   S704_WELD_BUFF_DATA31.RBT2_BT_CODE_NO := W#16#0;
   S704_WELD_BUFF_DATA31.RBT2_WELD_COUNT := W#16#0;
   S704_WELD_BUFF_DATA31.RBT3_BT_CODE_NO := W#16#0;
   S704_WELD_BUFF_DATA31.RBT3_WELD_COUNT := W#16#0;
   S704_WELD_BUFF_DATA31.RBT4_BT_CODE_NO := W#16#0;
   S704_WELD_BUFF_DATA31.RBT4_WELD_COUNT := W#16#0;
   S704_WELD_BUFF_DATA31.RBT5_BT_CODE_NO := W#16#0;
   S704_WELD_BUFF_DATA31.RBT5_WELD_COUNT := W#16#0;
   S704_WELD_BUFF_DATA31.RBT6_BT_CODE_NO := W#16#0;
   S704_WELD_BUFF_DATA31.RBT6_WELD_COUNT := W#16#0;
   S704_WELD_BUFF_DATA31.RBT7_BT_CODE_NO := W#16#0;
   S704_WELD_BUFF_DATA31.RBT7_WELD_COUNT := W#16#0;
   S704_WELD_BUFF_DATA31.RBT8_BT_CODE_NO := W#16#0;
   S704_WELD_BUFF_DATA31.RBT8_WELD_COUNT := W#16#0;
   S704_WELD_BUFF_DATA31.RBT9_BT_CODE_NO := W#16#0;
   S704_WELD_BUFF_DATA31.RBT9_WELD_COUNT := W#16#0;
   S704_WELD_BUFF_DATA31.RBT10_BT_CODE_NO := W#16#0;
   S704_WELD_BUFF_DATA31.RBT10_WELD_COUNT := W#16#0;
   S704_WELD_BUFF_DATA31.RBT11_BT_CODE_NO := W#16#0;
   S704_WELD_BUFF_DATA31.RBT11_WELD_COUNT := W#16#0;
   S704_WELD_BUFF_DATA31.RBT12_BT_CODE_NO := W#16#0;
   S704_WELD_BUFF_DATA31.RBT12_WELD_COUNT := W#16#0;
   S704_WELD_BUFF_DATA31.RBT13_BT_CODE_NO := W#16#0;
   S704_WELD_BUFF_DATA31.RBT13_WELD_COUNT := W#16#0;
   S704_WELD_BUFF_DATA31.RBT14_BT_CODE_NO := W#16#0;
   S704_WELD_BUFF_DATA31.RBT14_WELD_COUNT := W#16#0;
   S704_WELD_BUFF_DATA31.RBT15_BT_CODE_NO := W#16#0;
   S704_WELD_BUFF_DATA31.RBT15_WELD_COUNT := W#16#0;
   S704_WELD_BUFF_DATA31.RBT16_BT_CODE_NO := W#16#0;
   S704_WELD_BUFF_DATA31.RBT16_WELD_COUNT := W#16#0;
   S704_WELD_BUFF_DATA31.RBT17_BT_CODE_NO := W#16#0;
   S704_WELD_BUFF_DATA31.RBT17_WELD_COUNT := W#16#0;
   S704_WELD_BUFF_DATA31.RBT18_BT_CODE_NO := W#16#0;
   S704_WELD_BUFF_DATA31.RBT18_WELD_COUNT := W#16#0;
   S704_WELD_BUFF_DATA31.RBT19_BT_CODE_NO := W#16#0;
   S704_WELD_BUFF_DATA31.RBT19_WELD_COUNT := W#16#0;
   S704_WELD_BUFF_DATA31.RBT20_BT_CODE_NO := W#16#0;
   S704_WELD_BUFF_DATA31.RBT20_WELD_COUNT := W#16#0;
   S704_WELD_BUFF_DATA31.RBT21_BT_CODE_NO := W#16#0;
   S704_WELD_BUFF_DATA31.RBT21_WELD_COUNT := W#16#0;
   S704_WELD_BUFF_DATA31.RBT22_BT_CODE_NO := W#16#0;
   S704_WELD_BUFF_DATA31.RBT22_WELD_COUNT := W#16#0;
   S704_WELD_BUFF_DATA31.RBT23_BT_CODE_NO := W#16#0;
   S704_WELD_BUFF_DATA31.RBT23_WELD_COUNT := W#16#0;
   S704_WELD_BUFF_DATA31.RBT24_BT_CODE_NO := W#16#0;
   S704_WELD_BUFF_DATA31.RBT24_WELD_COUNT := W#16#0;
   S704_WELD_BUFF_DATA31.WELD_DETERMINES_RESULT := W#16#0;
   S704_WELD_BUFF_DATA31.WELD_CHECK_SUM := W#16#0;
   S704_WELD_BUFF_DATA31.SPARE1 := W#16#0;
   S704_WELD_BUFF_DATA41.STATION_MAIN := W#16#0;
   S704_WELD_BUFF_DATA41.DISTINCTION_LH_RH := W#16#0;
   S704_WELD_BUFF_DATA41.STAION_NUMBER := W#16#0;
   S704_WELD_BUFF_DATA41.VIN_NUMBER1 := W#16#0;
   S704_WELD_BUFF_DATA41.VIN_NUMBER2 := W#16#0;
   S704_WELD_BUFF_DATA41.VIN_NUMBER3 := W#16#0;
   S704_WELD_BUFF_DATA41.VIN_NUMBER4 := W#16#0;
   S704_WELD_BUFF_DATA41.SEQ_NUMBER1 := W#16#0;
   S704_WELD_BUFF_DATA41.SEQ_NUMBER2 := W#16#0;
   S704_WELD_BUFF_DATA41.RBT1_BT_CODE_NO := W#16#0;
   S704_WELD_BUFF_DATA41.RBT1_WELD_COUNT := W#16#0;
   S704_WELD_BUFF_DATA41.RBT2_BT_CODE_NO := W#16#0;
   S704_WELD_BUFF_DATA41.RBT2_WELD_COUNT := W#16#0;
   S704_WELD_BUFF_DATA41.RBT3_BT_CODE_NO := W#16#0;
   S704_WELD_BUFF_DATA41.RBT3_WELD_COUNT := W#16#0;
   S704_WELD_BUFF_DATA41.RBT4_BT_CODE_NO := W#16#0;
   S704_WELD_BUFF_DATA41.RBT4_WELD_COUNT := W#16#0;
   S704_WELD_BUFF_DATA41.RBT5_BT_CODE_NO := W#16#0;
   S704_WELD_BUFF_DATA41.RBT5_WELD_COUNT := W#16#0;
   S704_WELD_BUFF_DATA41.RBT6_BT_CODE_NO := W#16#0;
   S704_WELD_BUFF_DATA41.RBT6_WELD_COUNT := W#16#0;
   S704_WELD_BUFF_DATA41.RBT7_BT_CODE_NO := W#16#0;
   S704_WELD_BUFF_DATA41.RBT7_WELD_COUNT := W#16#0;
   S704_WELD_BUFF_DATA41.RBT8_BT_CODE_NO := W#16#0;
   S704_WELD_BUFF_DATA41.RBT8_WELD_COUNT := W#16#0;
   S704_WELD_BUFF_DATA41.RBT9_BT_CODE_NO := W#16#0;
   S704_WELD_BUFF_DATA41.RBT9_WELD_COUNT := W#16#0;
   S704_WELD_BUFF_DATA41.RBT10_BT_CODE_NO := W#16#0;
   S704_WELD_BUFF_DATA41.RBT10_WELD_COUNT := W#16#0;
   S704_WELD_BUFF_DATA41.RBT11_BT_CODE_NO := W#16#0;
   S704_WELD_BUFF_DATA41.RBT11_WELD_COUNT := W#16#0;
   S704_WELD_BUFF_DATA41.RBT12_BT_CODE_NO := W#16#0;
   S704_WELD_BUFF_DATA41.RBT12_WELD_COUNT := W#16#0;
   S704_WELD_BUFF_DATA41.RBT13_BT_CODE_NO := W#16#0;
   S704_WELD_BUFF_DATA41.RBT13_WELD_COUNT := W#16#0;
   S704_WELD_BUFF_DATA41.RBT14_BT_CODE_NO := W#16#0;
   S704_WELD_BUFF_DATA41.RBT14_WELD_COUNT := W#16#0;
   S704_WELD_BUFF_DATA41.RBT15_BT_CODE_NO := W#16#0;
   S704_WELD_BUFF_DATA41.RBT15_WELD_COUNT := W#16#0;
   S704_WELD_BUFF_DATA41.RBT16_BT_CODE_NO := W#16#0;
   S704_WELD_BUFF_DATA41.RBT16_WELD_COUNT := W#16#0;
   S704_WELD_BUFF_DATA41.RBT17_BT_CODE_NO := W#16#0;
   S704_WELD_BUFF_DATA41.RBT17_WELD_COUNT := W#16#0;
   S704_WELD_BUFF_DATA41.RBT18_BT_CODE_NO := W#16#0;
   S704_WELD_BUFF_DATA41.RBT18_WELD_COUNT := W#16#0;
   S704_WELD_BUFF_DATA41.RBT19_BT_CODE_NO := W#16#0;
   S704_WELD_BUFF_DATA41.RBT19_WELD_COUNT := W#16#0;
   S704_WELD_BUFF_DATA41.RBT20_BT_CODE_NO := W#16#0;
   S704_WELD_BUFF_DATA41.RBT20_WELD_COUNT := W#16#0;
   S704_WELD_BUFF_DATA41.RBT21_BT_CODE_NO := W#16#0;
   S704_WELD_BUFF_DATA41.RBT21_WELD_COUNT := W#16#0;
   S704_WELD_BUFF_DATA41.RBT22_BT_CODE_NO := W#16#0;
   S704_WELD_BUFF_DATA41.RBT22_WELD_COUNT := W#16#0;
   S704_WELD_BUFF_DATA41.RBT23_BT_CODE_NO := W#16#0;
   S704_WELD_BUFF_DATA41.RBT23_WELD_COUNT := W#16#0;
   S704_WELD_BUFF_DATA41.RBT24_BT_CODE_NO := W#16#0;
   S704_WELD_BUFF_DATA41.RBT24_WELD_COUNT := W#16#0;
   S704_WELD_BUFF_DATA41.WELD_DETERMINES_RESULT := W#16#0;
   S704_WELD_BUFF_DATA41.WELD_CHECK_SUM := W#16#0;
   S704_WELD_BUFF_DATA41.SPARE1 := W#16#0;
   S704_WELD_BUFF_DATA51.STATION_MAIN := W#16#0;
   S704_WELD_BUFF_DATA51.DISTINCTION_LH_RH := W#16#0;
   S704_WELD_BUFF_DATA51.STAION_NUMBER := W#16#0;
   S704_WELD_BUFF_DATA51.VIN_NUMBER1 := W#16#0;
   S704_WELD_BUFF_DATA51.VIN_NUMBER2 := W#16#0;
   S704_WELD_BUFF_DATA51.VIN_NUMBER3 := W#16#0;
   S704_WELD_BUFF_DATA51.VIN_NUMBER4 := W#16#0;
   S704_WELD_BUFF_DATA51.SEQ_NUMBER1 := W#16#0;
   S704_WELD_BUFF_DATA51.SEQ_NUMBER2 := W#16#0;
   S704_WELD_BUFF_DATA51.RBT1_BT_CODE_NO := W#16#0;
   S704_WELD_BUFF_DATA51.RBT1_WELD_COUNT := W#16#0;
   S704_WELD_BUFF_DATA51.RBT2_BT_CODE_NO := W#16#0;
   S704_WELD_BUFF_DATA51.RBT2_WELD_COUNT := W#16#0;
   S704_WELD_BUFF_DATA51.RBT3_BT_CODE_NO := W#16#0;
   S704_WELD_BUFF_DATA51.RBT3_WELD_COUNT := W#16#0;
   S704_WELD_BUFF_DATA51.RBT4_BT_CODE_NO := W#16#0;
   S704_WELD_BUFF_DATA51.RBT4_WELD_COUNT := W#16#0;
   S704_WELD_BUFF_DATA51.RBT5_BT_CODE_NO := W#16#0;
   S704_WELD_BUFF_DATA51.RBT5_WELD_COUNT := W#16#0;
   S704_WELD_BUFF_DATA51.RBT6_BT_CODE_NO := W#16#0;
   S704_WELD_BUFF_DATA51.RBT6_WELD_COUNT := W#16#0;
   S704_WELD_BUFF_DATA51.RBT7_BT_CODE_NO := W#16#0;
   S704_WELD_BUFF_DATA51.RBT7_WELD_COUNT := W#16#0;
   S704_WELD_BUFF_DATA51.RBT8_BT_CODE_NO := W#16#0;
   S704_WELD_BUFF_DATA51.RBT8_WELD_COUNT := W#16#0;
   S704_WELD_BUFF_DATA51.RBT9_BT_CODE_NO := W#16#0;
   S704_WELD_BUFF_DATA51.RBT9_WELD_COUNT := W#16#0;
   S704_WELD_BUFF_DATA51.RBT10_BT_CODE_NO := W#16#0;
   S704_WELD_BUFF_DATA51.RBT10_WELD_COUNT := W#16#0;
   S704_WELD_BUFF_DATA51.RBT11_BT_CODE_NO := W#16#0;
   S704_WELD_BUFF_DATA51.RBT11_WELD_COUNT := W#16#0;
   S704_WELD_BUFF_DATA51.RBT12_BT_CODE_NO := W#16#0;
   S704_WELD_BUFF_DATA51.RBT12_WELD_COUNT := W#16#0;
   S704_WELD_BUFF_DATA51.RBT13_BT_CODE_NO := W#16#0;
   S704_WELD_BUFF_DATA51.RBT13_WELD_COUNT := W#16#0;
   S704_WELD_BUFF_DATA51.RBT14_BT_CODE_NO := W#16#0;
   S704_WELD_BUFF_DATA51.RBT14_WELD_COUNT := W#16#0;
   S704_WELD_BUFF_DATA51.RBT15_BT_CODE_NO := W#16#0;
   S704_WELD_BUFF_DATA51.RBT15_WELD_COUNT := W#16#0;
   S704_WELD_BUFF_DATA51.RBT16_BT_CODE_NO := W#16#0;
   S704_WELD_BUFF_DATA51.RBT16_WELD_COUNT := W#16#0;
   S704_WELD_BUFF_DATA51.RBT17_BT_CODE_NO := W#16#0;
   S704_WELD_BUFF_DATA51.RBT17_WELD_COUNT := W#16#0;
   S704_WELD_BUFF_DATA51.RBT18_BT_CODE_NO := W#16#0;
   S704_WELD_BUFF_DATA51.RBT18_WELD_COUNT := W#16#0;
   S704_WELD_BUFF_DATA51.RBT19_BT_CODE_NO := W#16#0;
   S704_WELD_BUFF_DATA51.RBT19_WELD_COUNT := W#16#0;
   S704_WELD_BUFF_DATA51.RBT20_BT_CODE_NO := W#16#0;
   S704_WELD_BUFF_DATA51.RBT20_WELD_COUNT := W#16#0;
   S704_WELD_BUFF_DATA51.RBT21_BT_CODE_NO := W#16#0;
   S704_WELD_BUFF_DATA51.RBT21_WELD_COUNT := W#16#0;
   S704_WELD_BUFF_DATA51.RBT22_BT_CODE_NO := W#16#0;
   S704_WELD_BUFF_DATA51.RBT22_WELD_COUNT := W#16#0;
   S704_WELD_BUFF_DATA51.RBT23_BT_CODE_NO := W#16#0;
   S704_WELD_BUFF_DATA51.RBT23_WELD_COUNT := W#16#0;
   S704_WELD_BUFF_DATA51.RBT24_BT_CODE_NO := W#16#0;
   S704_WELD_BUFF_DATA51.RBT24_WELD_COUNT := W#16#0;
   S704_WELD_BUFF_DATA51.WELD_DETERMINES_RESULT := W#16#0;
   S704_WELD_BUFF_DATA51.WELD_CHECK_SUM := W#16#0;
   S704_WELD_BUFF_DATA51.SPARE1 := W#16#0;
   S704_WELD_BUFF_DATA61.STATION_MAIN := W#16#0;
   S704_WELD_BUFF_DATA61.DISTINCTION_LH_RH := W#16#0;
   S704_WELD_BUFF_DATA61.STAION_NUMBER := W#16#0;
   S704_WELD_BUFF_DATA61.VIN_NUMBER1 := W#16#0;
   S704_WELD_BUFF_DATA61.VIN_NUMBER2 := W#16#0;
   S704_WELD_BUFF_DATA61.VIN_NUMBER3 := W#16#0;
   S704_WELD_BUFF_DATA61.VIN_NUMBER4 := W#16#0;
   S704_WELD_BUFF_DATA61.SEQ_NUMBER1 := W#16#0;
   S704_WELD_BUFF_DATA61.SEQ_NUMBER2 := W#16#0;
   S704_WELD_BUFF_DATA61.RBT1_BT_CODE_NO := W#16#0;
   S704_WELD_BUFF_DATA61.RBT1_WELD_COUNT := W#16#0;
   S704_WELD_BUFF_DATA61.RBT2_BT_CODE_NO := W#16#0;
   S704_WELD_BUFF_DATA61.RBT2_WELD_COUNT := W#16#0;
   S704_WELD_BUFF_DATA61.RBT3_BT_CODE_NO := W#16#0;
   S704_WELD_BUFF_DATA61.RBT3_WELD_COUNT := W#16#0;
   S704_WELD_BUFF_DATA61.RBT4_BT_CODE_NO := W#16#0;
   S704_WELD_BUFF_DATA61.RBT4_WELD_COUNT := W#16#0;
   S704_WELD_BUFF_DATA61.RBT5_BT_CODE_NO := W#16#0;
   S704_WELD_BUFF_DATA61.RBT5_WELD_COUNT := W#16#0;
   S704_WELD_BUFF_DATA61.RBT6_BT_CODE_NO := W#16#0;
   S704_WELD_BUFF_DATA61.RBT6_WELD_COUNT := W#16#0;
   S704_WELD_BUFF_DATA61.RBT7_BT_CODE_NO := W#16#0;
   S704_WELD_BUFF_DATA61.RBT7_WELD_COUNT := W#16#0;
   S704_WELD_BUFF_DATA61.RBT8_BT_CODE_NO := W#16#0;
   S704_WELD_BUFF_DATA61.RBT8_WELD_COUNT := W#16#0;
   S704_WELD_BUFF_DATA61.RBT9_BT_CODE_NO := W#16#0;
   S704_WELD_BUFF_DATA61.RBT9_WELD_COUNT := W#16#0;
   S704_WELD_BUFF_DATA61.RBT10_BT_CODE_NO := W#16#0;
   S704_WELD_BUFF_DATA61.RBT10_WELD_COUNT := W#16#0;
   S704_WELD_BUFF_DATA61.RBT11_BT_CODE_NO := W#16#0;
   S704_WELD_BUFF_DATA61.RBT11_WELD_COUNT := W#16#0;
   S704_WELD_BUFF_DATA61.RBT12_BT_CODE_NO := W#16#0;
   S704_WELD_BUFF_DATA61.RBT12_WELD_COUNT := W#16#0;
   S704_WELD_BUFF_DATA61.RBT13_BT_CODE_NO := W#16#0;
   S704_WELD_BUFF_DATA61.RBT13_WELD_COUNT := W#16#0;
   S704_WELD_BUFF_DATA61.RBT14_BT_CODE_NO := W#16#0;
   S704_WELD_BUFF_DATA61.RBT14_WELD_COUNT := W#16#0;
   S704_WELD_BUFF_DATA61.RBT15_BT_CODE_NO := W#16#0;
   S704_WELD_BUFF_DATA61.RBT15_WELD_COUNT := W#16#0;
   S704_WELD_BUFF_DATA61.RBT16_BT_CODE_NO := W#16#0;
   S704_WELD_BUFF_DATA61.RBT16_WELD_COUNT := W#16#0;
   S704_WELD_BUFF_DATA61.RBT17_BT_CODE_NO := W#16#0;
   S704_WELD_BUFF_DATA61.RBT17_WELD_COUNT := W#16#0;
   S704_WELD_BUFF_DATA61.RBT18_BT_CODE_NO := W#16#0;
   S704_WELD_BUFF_DATA61.RBT18_WELD_COUNT := W#16#0;
   S704_WELD_BUFF_DATA61.RBT19_BT_CODE_NO := W#16#0;
   S704_WELD_BUFF_DATA61.RBT19_WELD_COUNT := W#16#0;
   S704_WELD_BUFF_DATA61.RBT20_BT_CODE_NO := W#16#0;
   S704_WELD_BUFF_DATA61.RBT20_WELD_COUNT := W#16#0;
   S704_WELD_BUFF_DATA61.RBT21_BT_CODE_NO := W#16#0;
   S704_WELD_BUFF_DATA61.RBT21_WELD_COUNT := W#16#0;
   S704_WELD_BUFF_DATA61.RBT22_BT_CODE_NO := W#16#0;
   S704_WELD_BUFF_DATA61.RBT22_WELD_COUNT := W#16#0;
   S704_WELD_BUFF_DATA61.RBT23_BT_CODE_NO := W#16#0;
   S704_WELD_BUFF_DATA61.RBT23_WELD_COUNT := W#16#0;
   S704_WELD_BUFF_DATA61.RBT24_BT_CODE_NO := W#16#0;
   S704_WELD_BUFF_DATA61.RBT24_WELD_COUNT := W#16#0;
   S704_WELD_BUFF_DATA61.WELD_DETERMINES_RESULT := W#16#0;
   S704_WELD_BUFF_DATA61.WELD_CHECK_SUM := W#16#0;
   S704_WELD_BUFF_DATA61.SPARE1 := W#16#0;
   S704_WELD_BUFF_DATA71.STATION_MAIN := W#16#0;
   S704_WELD_BUFF_DATA71.DISTINCTION_LH_RH := W#16#0;
   S704_WELD_BUFF_DATA71.STAION_NUMBER := W#16#0;
   S704_WELD_BUFF_DATA71.VIN_NUMBER1 := W#16#0;
   S704_WELD_BUFF_DATA71.VIN_NUMBER2 := W#16#0;
   S704_WELD_BUFF_DATA71.VIN_NUMBER3 := W#16#0;
   S704_WELD_BUFF_DATA71.VIN_NUMBER4 := W#16#0;
   S704_WELD_BUFF_DATA71.SEQ_NUMBER1 := W#16#0;
   S704_WELD_BUFF_DATA71.SEQ_NUMBER2 := W#16#0;
   S704_WELD_BUFF_DATA71.RBT1_BT_CODE_NO := W#16#0;
   S704_WELD_BUFF_DATA71.RBT1_WELD_COUNT := W#16#0;
   S704_WELD_BUFF_DATA71.RBT2_BT_CODE_NO := W#16#0;
   S704_WELD_BUFF_DATA71.RBT2_WELD_COUNT := W#16#0;
   S704_WELD_BUFF_DATA71.RBT3_BT_CODE_NO := W#16#0;
   S704_WELD_BUFF_DATA71.RBT3_WELD_COUNT := W#16#0;
   S704_WELD_BUFF_DATA71.RBT4_BT_CODE_NO := W#16#0;
   S704_WELD_BUFF_DATA71.RBT4_WELD_COUNT := W#16#0;
   S704_WELD_BUFF_DATA71.RBT5_BT_CODE_NO := W#16#0;
   S704_WELD_BUFF_DATA71.RBT5_WELD_COUNT := W#16#0;
   S704_WELD_BUFF_DATA71.RBT6_BT_CODE_NO := W#16#0;
   S704_WELD_BUFF_DATA71.RBT6_WELD_COUNT := W#16#0;
   S704_WELD_BUFF_DATA71.RBT7_BT_CODE_NO := W#16#0;
   S704_WELD_BUFF_DATA71.RBT7_WELD_COUNT := W#16#0;
   S704_WELD_BUFF_DATA71.RBT8_BT_CODE_NO := W#16#0;
   S704_WELD_BUFF_DATA71.RBT8_WELD_COUNT := W#16#0;
   S704_WELD_BUFF_DATA71.RBT9_BT_CODE_NO := W#16#0;
   S704_WELD_BUFF_DATA71.RBT9_WELD_COUNT := W#16#0;
   S704_WELD_BUFF_DATA71.RBT10_BT_CODE_NO := W#16#0;
   S704_WELD_BUFF_DATA71.RBT10_WELD_COUNT := W#16#0;
   S704_WELD_BUFF_DATA71.RBT11_BT_CODE_NO := W#16#0;
   S704_WELD_BUFF_DATA71.RBT11_WELD_COUNT := W#16#0;
   S704_WELD_BUFF_DATA71.RBT12_BT_CODE_NO := W#16#0;
   S704_WELD_BUFF_DATA71.RBT12_WELD_COUNT := W#16#0;
   S704_WELD_BUFF_DATA71.RBT13_BT_CODE_NO := W#16#0;
   S704_WELD_BUFF_DATA71.RBT13_WELD_COUNT := W#16#0;
   S704_WELD_BUFF_DATA71.RBT14_BT_CODE_NO := W#16#0;
   S704_WELD_BUFF_DATA71.RBT14_WELD_COUNT := W#16#0;
   S704_WELD_BUFF_DATA71.RBT15_BT_CODE_NO := W#16#0;
   S704_WELD_BUFF_DATA71.RBT15_WELD_COUNT := W#16#0;
   S704_WELD_BUFF_DATA71.RBT16_BT_CODE_NO := W#16#0;
   S704_WELD_BUFF_DATA71.RBT16_WELD_COUNT := W#16#0;
   S704_WELD_BUFF_DATA71.RBT17_BT_CODE_NO := W#16#0;
   S704_WELD_BUFF_DATA71.RBT17_WELD_COUNT := W#16#0;
   S704_WELD_BUFF_DATA71.RBT18_BT_CODE_NO := W#16#0;
   S704_WELD_BUFF_DATA71.RBT18_WELD_COUNT := W#16#0;
   S704_WELD_BUFF_DATA71.RBT19_BT_CODE_NO := W#16#0;
   S704_WELD_BUFF_DATA71.RBT19_WELD_COUNT := W#16#0;
   S704_WELD_BUFF_DATA71.RBT20_BT_CODE_NO := W#16#0;
   S704_WELD_BUFF_DATA71.RBT20_WELD_COUNT := W#16#0;
   S704_WELD_BUFF_DATA71.RBT21_BT_CODE_NO := W#16#0;
   S704_WELD_BUFF_DATA71.RBT21_WELD_COUNT := W#16#0;
   S704_WELD_BUFF_DATA71.RBT22_BT_CODE_NO := W#16#0;
   S704_WELD_BUFF_DATA71.RBT22_WELD_COUNT := W#16#0;
   S704_WELD_BUFF_DATA71.RBT23_BT_CODE_NO := W#16#0;
   S704_WELD_BUFF_DATA71.RBT23_WELD_COUNT := W#16#0;
   S704_WELD_BUFF_DATA71.RBT24_BT_CODE_NO := W#16#0;
   S704_WELD_BUFF_DATA71.RBT24_WELD_COUNT := W#16#0;
   S704_WELD_BUFF_DATA71.WELD_DETERMINES_RESULT := W#16#0;
   S704_WELD_BUFF_DATA71.WELD_CHECK_SUM := W#16#0;
   S704_WELD_BUFF_DATA71.SPARE1 := W#16#0;
   S704_WELD_BUFF_DATA81.STATION_MAIN := W#16#0;
   S704_WELD_BUFF_DATA81.DISTINCTION_LH_RH := W#16#0;
   S704_WELD_BUFF_DATA81.STAION_NUMBER := W#16#0;
   S704_WELD_BUFF_DATA81.VIN_NUMBER1 := W#16#0;
   S704_WELD_BUFF_DATA81.VIN_NUMBER2 := W#16#0;
   S704_WELD_BUFF_DATA81.VIN_NUMBER3 := W#16#0;
   S704_WELD_BUFF_DATA81.VIN_NUMBER4 := W#16#0;
   S704_WELD_BUFF_DATA81.SEQ_NUMBER1 := W#16#0;
   S704_WELD_BUFF_DATA81.SEQ_NUMBER2 := W#16#0;
   S704_WELD_BUFF_DATA81.RBT1_BT_CODE_NO := W#16#0;
   S704_WELD_BUFF_DATA81.RBT1_WELD_COUNT := W#16#0;
   S704_WELD_BUFF_DATA81.RBT2_BT_CODE_NO := W#16#0;
   S704_WELD_BUFF_DATA81.RBT2_WELD_COUNT := W#16#0;
   S704_WELD_BUFF_DATA81.RBT3_BT_CODE_NO := W#16#0;
   S704_WELD_BUFF_DATA81.RBT3_WELD_COUNT := W#16#0;
   S704_WELD_BUFF_DATA81.RBT4_BT_CODE_NO := W#16#0;
   S704_WELD_BUFF_DATA81.RBT4_WELD_COUNT := W#16#0;
   S704_WELD_BUFF_DATA81.RBT5_BT_CODE_NO := W#16#0;
   S704_WELD_BUFF_DATA81.RBT5_WELD_COUNT := W#16#0;
   S704_WELD_BUFF_DATA81.RBT6_BT_CODE_NO := W#16#0;
   S704_WELD_BUFF_DATA81.RBT6_WELD_COUNT := W#16#0;
   S704_WELD_BUFF_DATA81.RBT7_BT_CODE_NO := W#16#0;
   S704_WELD_BUFF_DATA81.RBT7_WELD_COUNT := W#16#0;
   S704_WELD_BUFF_DATA81.RBT8_BT_CODE_NO := W#16#0;
   S704_WELD_BUFF_DATA81.RBT8_WELD_COUNT := W#16#0;
   S704_WELD_BUFF_DATA81.RBT9_BT_CODE_NO := W#16#0;
   S704_WELD_BUFF_DATA81.RBT9_WELD_COUNT := W#16#0;
   S704_WELD_BUFF_DATA81.RBT10_BT_CODE_NO := W#16#0;
   S704_WELD_BUFF_DATA81.RBT10_WELD_COUNT := W#16#0;
   S704_WELD_BUFF_DATA81.RBT11_BT_CODE_NO := W#16#0;
   S704_WELD_BUFF_DATA81.RBT11_WELD_COUNT := W#16#0;
   S704_WELD_BUFF_DATA81.RBT12_BT_CODE_NO := W#16#0;
   S704_WELD_BUFF_DATA81.RBT12_WELD_COUNT := W#16#0;
   S704_WELD_BUFF_DATA81.RBT13_BT_CODE_NO := W#16#0;
   S704_WELD_BUFF_DATA81.RBT13_WELD_COUNT := W#16#0;
   S704_WELD_BUFF_DATA81.RBT14_BT_CODE_NO := W#16#0;
   S704_WELD_BUFF_DATA81.RBT14_WELD_COUNT := W#16#0;
   S704_WELD_BUFF_DATA81.RBT15_BT_CODE_NO := W#16#0;
   S704_WELD_BUFF_DATA81.RBT15_WELD_COUNT := W#16#0;
   S704_WELD_BUFF_DATA81.RBT16_BT_CODE_NO := W#16#0;
   S704_WELD_BUFF_DATA81.RBT16_WELD_COUNT := W#16#0;
   S704_WELD_BUFF_DATA81.RBT17_BT_CODE_NO := W#16#0;
   S704_WELD_BUFF_DATA81.RBT17_WELD_COUNT := W#16#0;
   S704_WELD_BUFF_DATA81.RBT18_BT_CODE_NO := W#16#0;
   S704_WELD_BUFF_DATA81.RBT18_WELD_COUNT := W#16#0;
   S704_WELD_BUFF_DATA81.RBT19_BT_CODE_NO := W#16#0;
   S704_WELD_BUFF_DATA81.RBT19_WELD_COUNT := W#16#0;
   S704_WELD_BUFF_DATA81.RBT20_BT_CODE_NO := W#16#0;
   S704_WELD_BUFF_DATA81.RBT20_WELD_COUNT := W#16#0;
   S704_WELD_BUFF_DATA81.RBT21_BT_CODE_NO := W#16#0;
   S704_WELD_BUFF_DATA81.RBT21_WELD_COUNT := W#16#0;
   S704_WELD_BUFF_DATA81.RBT22_BT_CODE_NO := W#16#0;
   S704_WELD_BUFF_DATA81.RBT22_WELD_COUNT := W#16#0;
   S704_WELD_BUFF_DATA81.RBT23_BT_CODE_NO := W#16#0;
   S704_WELD_BUFF_DATA81.RBT23_WELD_COUNT := W#16#0;
   S704_WELD_BUFF_DATA81.RBT24_BT_CODE_NO := W#16#0;
   S704_WELD_BUFF_DATA81.RBT24_WELD_COUNT := W#16#0;
   S704_WELD_BUFF_DATA81.WELD_DETERMINES_RESULT := W#16#0;
   S704_WELD_BUFF_DATA81.WELD_CHECK_SUM := W#16#0;
   S704_WELD_BUFF_DATA81.SPARE1 := W#16#0;
   S704_WELD_BUFF_DATA91.STATION_MAIN := W#16#0;
   S704_WELD_BUFF_DATA91.DISTINCTION_LH_RH := W#16#0;
   S704_WELD_BUFF_DATA91.STAION_NUMBER := W#16#0;
   S704_WELD_BUFF_DATA91.VIN_NUMBER1 := W#16#0;
   S704_WELD_BUFF_DATA91.VIN_NUMBER2 := W#16#0;
   S704_WELD_BUFF_DATA91.VIN_NUMBER3 := W#16#0;
   S704_WELD_BUFF_DATA91.VIN_NUMBER4 := W#16#0;
   S704_WELD_BUFF_DATA91.SEQ_NUMBER1 := W#16#0;
   S704_WELD_BUFF_DATA91.SEQ_NUMBER2 := W#16#0;
   S704_WELD_BUFF_DATA91.RBT1_BT_CODE_NO := W#16#0;
   S704_WELD_BUFF_DATA91.RBT1_WELD_COUNT := W#16#0;
   S704_WELD_BUFF_DATA91.RBT2_BT_CODE_NO := W#16#0;
   S704_WELD_BUFF_DATA91.RBT2_WELD_COUNT := W#16#0;
   S704_WELD_BUFF_DATA91.RBT3_BT_CODE_NO := W#16#0;
   S704_WELD_BUFF_DATA91.RBT3_WELD_COUNT := W#16#0;
   S704_WELD_BUFF_DATA91.RBT4_BT_CODE_NO := W#16#0;
   S704_WELD_BUFF_DATA91.RBT4_WELD_COUNT := W#16#0;
   S704_WELD_BUFF_DATA91.RBT5_BT_CODE_NO := W#16#0;
   S704_WELD_BUFF_DATA91.RBT5_WELD_COUNT := W#16#0;
   S704_WELD_BUFF_DATA91.RBT6_BT_CODE_NO := W#16#0;
   S704_WELD_BUFF_DATA91.RBT6_WELD_COUNT := W#16#0;
   S704_WELD_BUFF_DATA91.RBT7_BT_CODE_NO := W#16#0;
   S704_WELD_BUFF_DATA91.RBT7_WELD_COUNT := W#16#0;
   S704_WELD_BUFF_DATA91.RBT8_BT_CODE_NO := W#16#0;
   S704_WELD_BUFF_DATA91.RBT8_WELD_COUNT := W#16#0;
   S704_WELD_BUFF_DATA91.RBT9_BT_CODE_NO := W#16#0;
   S704_WELD_BUFF_DATA91.RBT9_WELD_COUNT := W#16#0;
   S704_WELD_BUFF_DATA91.RBT10_BT_CODE_NO := W#16#0;
   S704_WELD_BUFF_DATA91.RBT10_WELD_COUNT := W#16#0;
   S704_WELD_BUFF_DATA91.RBT11_BT_CODE_NO := W#16#0;
   S704_WELD_BUFF_DATA91.RBT11_WELD_COUNT := W#16#0;
   S704_WELD_BUFF_DATA91.RBT12_BT_CODE_NO := W#16#0;
   S704_WELD_BUFF_DATA91.RBT12_WELD_COUNT := W#16#0;
   S704_WELD_BUFF_DATA91.RBT13_BT_CODE_NO := W#16#0;
   S704_WELD_BUFF_DATA91.RBT13_WELD_COUNT := W#16#0;
   S704_WELD_BUFF_DATA91.RBT14_BT_CODE_NO := W#16#0;
   S704_WELD_BUFF_DATA91.RBT14_WELD_COUNT := W#16#0;
   S704_WELD_BUFF_DATA91.RBT15_BT_CODE_NO := W#16#0;
   S704_WELD_BUFF_DATA91.RBT15_WELD_COUNT := W#16#0;
   S704_WELD_BUFF_DATA91.RBT16_BT_CODE_NO := W#16#0;
   S704_WELD_BUFF_DATA91.RBT16_WELD_COUNT := W#16#0;
   S704_WELD_BUFF_DATA91.RBT17_BT_CODE_NO := W#16#0;
   S704_WELD_BUFF_DATA91.RBT17_WELD_COUNT := W#16#0;
   S704_WELD_BUFF_DATA91.RBT18_BT_CODE_NO := W#16#0;
   S704_WELD_BUFF_DATA91.RBT18_WELD_COUNT := W#16#0;
   S704_WELD_BUFF_DATA91.RBT19_BT_CODE_NO := W#16#0;
   S704_WELD_BUFF_DATA91.RBT19_WELD_COUNT := W#16#0;
   S704_WELD_BUFF_DATA91.RBT20_BT_CODE_NO := W#16#0;
   S704_WELD_BUFF_DATA91.RBT20_WELD_COUNT := W#16#0;
   S704_WELD_BUFF_DATA91.RBT21_BT_CODE_NO := W#16#0;
   S704_WELD_BUFF_DATA91.RBT21_WELD_COUNT := W#16#0;
   S704_WELD_BUFF_DATA91.RBT22_BT_CODE_NO := W#16#0;
   S704_WELD_BUFF_DATA91.RBT22_WELD_COUNT := W#16#0;
   S704_WELD_BUFF_DATA91.RBT23_BT_CODE_NO := W#16#0;
   S704_WELD_BUFF_DATA91.RBT23_WELD_COUNT := W#16#0;
   S704_WELD_BUFF_DATA91.RBT24_BT_CODE_NO := W#16#0;
   S704_WELD_BUFF_DATA91.RBT24_WELD_COUNT := W#16#0;
   S704_WELD_BUFF_DATA91.WELD_DETERMINES_RESULT := W#16#0;
   S704_WELD_BUFF_DATA91.WELD_CHECK_SUM := W#16#0;
   S704_WELD_BUFF_DATA91.SPARE1 := W#16#0;
   S704_WELD_BUFF_DATA101.STATION_MAIN := W#16#0;
   S704_WELD_BUFF_DATA101.DISTINCTION_LH_RH := W#16#0;
   S704_WELD_BUFF_DATA101.STAION_NUMBER := W#16#0;
   S704_WELD_BUFF_DATA101.VIN_NUMBER1 := W#16#0;
   S704_WELD_BUFF_DATA101.VIN_NUMBER2 := W#16#0;
   S704_WELD_BUFF_DATA101.VIN_NUMBER3 := W#16#0;
   S704_WELD_BUFF_DATA101.VIN_NUMBER4 := W#16#0;
   S704_WELD_BUFF_DATA101.SEQ_NUMBER1 := W#16#0;
   S704_WELD_BUFF_DATA101.SEQ_NUMBER2 := W#16#0;
   S704_WELD_BUFF_DATA101.RBT1_BT_CODE_NO := W#16#0;
   S704_WELD_BUFF_DATA101.RBT1_WELD_COUNT := W#16#0;
   S704_WELD_BUFF_DATA101.RBT2_BT_CODE_NO := W#16#0;
   S704_WELD_BUFF_DATA101.RBT2_WELD_COUNT := W#16#0;
   S704_WELD_BUFF_DATA101.RBT3_BT_CODE_NO := W#16#0;
   S704_WELD_BUFF_DATA101.RBT3_WELD_COUNT := W#16#0;
   S704_WELD_BUFF_DATA101.RBT4_BT_CODE_NO := W#16#0;
   S704_WELD_BUFF_DATA101.RBT4_WELD_COUNT := W#16#0;
   S704_WELD_BUFF_DATA101.RBT5_BT_CODE_NO := W#16#0;
   S704_WELD_BUFF_DATA101.RBT5_WELD_COUNT := W#16#0;
   S704_WELD_BUFF_DATA101.RBT6_BT_CODE_NO := W#16#0;
   S704_WELD_BUFF_DATA101.RBT6_WELD_COUNT := W#16#0;
   S704_WELD_BUFF_DATA101.RBT7_BT_CODE_NO := W#16#0;
   S704_WELD_BUFF_DATA101.RBT7_WELD_COUNT := W#16#0;
   S704_WELD_BUFF_DATA101.RBT8_BT_CODE_NO := W#16#0;
   S704_WELD_BUFF_DATA101.RBT8_WELD_COUNT := W#16#0;
   S704_WELD_BUFF_DATA101.RBT9_BT_CODE_NO := W#16#0;
   S704_WELD_BUFF_DATA101.RBT9_WELD_COUNT := W#16#0;
   S704_WELD_BUFF_DATA101.RBT10_BT_CODE_NO := W#16#0;
   S704_WELD_BUFF_DATA101.RBT10_WELD_COUNT := W#16#0;
   S704_WELD_BUFF_DATA101.RBT11_BT_CODE_NO := W#16#0;
   S704_WELD_BUFF_DATA101.RBT11_WELD_COUNT := W#16#0;
   S704_WELD_BUFF_DATA101.RBT12_BT_CODE_NO := W#16#0;
   S704_WELD_BUFF_DATA101.RBT12_WELD_COUNT := W#16#0;
   S704_WELD_BUFF_DATA101.RBT13_BT_CODE_NO := W#16#0;
   S704_WELD_BUFF_DATA101.RBT13_WELD_COUNT := W#16#0;
   S704_WELD_BUFF_DATA101.RBT14_BT_CODE_NO := W#16#0;
   S704_WELD_BUFF_DATA101.RBT14_WELD_COUNT := W#16#0;
   S704_WELD_BUFF_DATA101.RBT15_BT_CODE_NO := W#16#0;
   S704_WELD_BUFF_DATA101.RBT15_WELD_COUNT := W#16#0;
   S704_WELD_BUFF_DATA101.RBT16_BT_CODE_NO := W#16#0;
   S704_WELD_BUFF_DATA101.RBT16_WELD_COUNT := W#16#0;
   S704_WELD_BUFF_DATA101.RBT17_BT_CODE_NO := W#16#0;
   S704_WELD_BUFF_DATA101.RBT17_WELD_COUNT := W#16#0;
   S704_WELD_BUFF_DATA101.RBT18_BT_CODE_NO := W#16#0;
   S704_WELD_BUFF_DATA101.RBT18_WELD_COUNT := W#16#0;
   S704_WELD_BUFF_DATA101.RBT19_BT_CODE_NO := W#16#0;
   S704_WELD_BUFF_DATA101.RBT19_WELD_COUNT := W#16#0;
   S704_WELD_BUFF_DATA101.RBT20_BT_CODE_NO := W#16#0;
   S704_WELD_BUFF_DATA101.RBT20_WELD_COUNT := W#16#0;
   S704_WELD_BUFF_DATA101.RBT21_BT_CODE_NO := W#16#0;
   S704_WELD_BUFF_DATA101.RBT21_WELD_COUNT := W#16#0;
   S704_WELD_BUFF_DATA101.RBT22_BT_CODE_NO := W#16#0;
   S704_WELD_BUFF_DATA101.RBT22_WELD_COUNT := W#16#0;
   S704_WELD_BUFF_DATA101.RBT23_BT_CODE_NO := W#16#0;
   S704_WELD_BUFF_DATA101.RBT23_WELD_COUNT := W#16#0;
   S704_WELD_BUFF_DATA101.RBT24_BT_CODE_NO := W#16#0;
   S704_WELD_BUFF_DATA101.RBT24_WELD_COUNT := W#16#0;
   S704_WELD_BUFF_DATA101.WELD_DETERMINES_RESULT := W#16#0;
   S704_WELD_BUFF_DATA101.WELD_CHECK_SUM := W#16#0;
   S704_WELD_BUFF_DATA101.SPARE1 := W#16#0;
END_DATA_BLOCK

DATA_BLOCK DB 45
TITLE =
VERSION : 0.1


  STRUCT
   STAT0 : ARRAY  [0 .. 99 ] OF WORD  := W#16#0;
   STAT01 : ARRAY  [0 .. 99 ] OF WORD  := W#16#0;
   STAT011 : ARRAY  [0 .. 99 ] OF WORD  := W#16#0;
  END_STRUCT ;
BEGIN
   STAT0[0] := W#16#0;
   STAT0[1] := W#16#0;
   STAT0[2] := W#16#0;
   STAT0[3] := W#16#0;
   STAT0[4] := W#16#0;
   STAT0[5] := W#16#0;
   STAT0[6] := W#16#0;
   STAT0[7] := W#16#0;
   STAT0[8] := W#16#0;
   STAT0[9] := W#16#0;
   STAT0[10] := W#16#0;
   STAT0[11] := W#16#0;
   STAT0[12] := W#16#0;
   STAT0[13] := W#16#0;
   STAT0[14] := W#16#0;
   STAT0[15] := W#16#0;
   STAT0[16] := W#16#0;
   STAT0[17] := W#16#0;
   STAT0[18] := W#16#0;
   STAT0[19] := W#16#0;
   STAT0[20] := W#16#0;
   STAT0[21] := W#16#0;
   STAT0[22] := W#16#0;
   STAT0[23] := W#16#0;
   STAT0[24] := W#16#0;
   STAT0[25] := W#16#0;
   STAT0[26] := W#16#0;
   STAT0[27] := W#16#0;
   STAT0[28] := W#16#0;
   STAT0[29] := W#16#0;
   STAT0[30] := W#16#0;
   STAT0[31] := W#16#0;
   STAT0[32] := W#16#0;
   STAT0[33] := W#16#0;
   STAT0[34] := W#16#0;
   STAT0[35] := W#16#0;
   STAT0[36] := W#16#0;
   STAT0[37] := W#16#0;
   STAT0[38] := W#16#0;
   STAT0[39] := W#16#0;
   STAT0[40] := W#16#0;
   STAT0[41] := W#16#0;
   STAT0[42] := W#16#0;
   STAT0[43] := W#16#0;
   STAT0[44] := W#16#0;
   STAT0[45] := W#16#0;
   STAT0[46] := W#16#0;
   STAT0[47] := W#16#0;
   STAT0[48] := W#16#0;
   STAT0[49] := W#16#0;
   STAT0[50] := W#16#0;
   STAT0[51] := W#16#0;
   STAT0[52] := W#16#0;
   STAT0[53] := W#16#0;
   STAT0[54] := W#16#0;
   STAT0[55] := W#16#0;
   STAT0[56] := W#16#0;
   STAT0[57] := W#16#0;
   STAT0[58] := W#16#0;
   STAT0[59] := W#16#0;
   STAT0[60] := W#16#0;
   STAT0[61] := W#16#0;
   STAT0[62] := W#16#0;
   STAT0[63] := W#16#0;
   STAT0[64] := W#16#0;
   STAT0[65] := W#16#0;
   STAT0[66] := W#16#0;
   STAT0[67] := W#16#0;
   STAT0[68] := W#16#0;
   STAT0[69] := W#16#0;
   STAT0[70] := W#16#0;
   STAT0[71] := W#16#0;
   STAT0[72] := W#16#0;
   STAT0[73] := W#16#0;
   STAT0[74] := W#16#0;
   STAT0[75] := W#16#0;
   STAT0[76] := W#16#0;
   STAT0[77] := W#16#0;
   STAT0[78] := W#16#0;
   STAT0[79] := W#16#0;
   STAT0[80] := W#16#0;
   STAT0[81] := W#16#0;
   STAT0[82] := W#16#0;
   STAT0[83] := W#16#0;
   STAT0[84] := W#16#0;
   STAT0[85] := W#16#0;
   STAT0[86] := W#16#0;
   STAT0[87] := W#16#0;
   STAT0[88] := W#16#0;
   STAT0[89] := W#16#0;
   STAT0[90] := W#16#0;
   STAT0[91] := W#16#0;
   STAT0[92] := W#16#0;
   STAT0[93] := W#16#0;
   STAT0[94] := W#16#0;
   STAT0[95] := W#16#0;
   STAT0[96] := W#16#0;
   STAT0[97] := W#16#0;
   STAT0[98] := W#16#0;
   STAT0[99] := W#16#0;
   STAT01[0] := W#16#0;
   STAT01[1] := W#16#0;
   STAT01[2] := W#16#0;
   STAT01[3] := W#16#0;
   STAT01[4] := W#16#0;
   STAT01[5] := W#16#0;
   STAT01[6] := W#16#0;
   STAT01[7] := W#16#0;
   STAT01[8] := W#16#0;
   STAT01[9] := W#16#0;
   STAT01[10] := W#16#0;
   STAT01[11] := W#16#0;
   STAT01[12] := W#16#0;
   STAT01[13] := W#16#0;
   STAT01[14] := W#16#0;
   STAT01[15] := W#16#0;
   STAT01[16] := W#16#0;
   STAT01[17] := W#16#0;
   STAT01[18] := W#16#0;
   STAT01[19] := W#16#0;
   STAT01[20] := W#16#0;
   STAT01[21] := W#16#0;
   STAT01[22] := W#16#0;
   STAT01[23] := W#16#0;
   STAT01[24] := W#16#0;
   STAT01[25] := W#16#0;
   STAT01[26] := W#16#0;
   STAT01[27] := W#16#0;
   STAT01[28] := W#16#0;
   STAT01[29] := W#16#0;
   STAT01[30] := W#16#0;
   STAT01[31] := W#16#0;
   STAT01[32] := W#16#0;
   STAT01[33] := W#16#0;
   STAT01[34] := W#16#0;
   STAT01[35] := W#16#0;
   STAT01[36] := W#16#0;
   STAT01[37] := W#16#0;
   STAT01[38] := W#16#0;
   STAT01[39] := W#16#0;
   STAT01[40] := W#16#0;
   STAT01[41] := W#16#0;
   STAT01[42] := W#16#0;
   STAT01[43] := W#16#0;
   STAT01[44] := W#16#0;
   STAT01[45] := W#16#0;
   STAT01[46] := W#16#0;
   STAT01[47] := W#16#0;
   STAT01[48] := W#16#0;
   STAT01[49] := W#16#0;
   STAT01[50] := W#16#0;
   STAT01[51] := W#16#0;
   STAT01[52] := W#16#0;
   STAT01[53] := W#16#0;
   STAT01[54] := W#16#0;
   STAT01[55] := W#16#0;
   STAT01[56] := W#16#0;
   STAT01[57] := W#16#0;
   STAT01[58] := W#16#0;
   STAT01[59] := W#16#0;
   STAT01[60] := W#16#0;
   STAT01[61] := W#16#0;
   STAT01[62] := W#16#0;
   STAT01[63] := W#16#0;
   STAT01[64] := W#16#0;
   STAT01[65] := W#16#0;
   STAT01[66] := W#16#0;
   STAT01[67] := W#16#0;
   STAT01[68] := W#16#0;
   STAT01[69] := W#16#0;
   STAT01[70] := W#16#0;
   STAT01[71] := W#16#0;
   STAT01[72] := W#16#0;
   STAT01[73] := W#16#0;
   STAT01[74] := W#16#0;
   STAT01[75] := W#16#0;
   STAT01[76] := W#16#0;
   STAT01[77] := W#16#0;
   STAT01[78] := W#16#0;
   STAT01[79] := W#16#0;
   STAT01[80] := W#16#0;
   STAT01[81] := W#16#0;
   STAT01[82] := W#16#0;
   STAT01[83] := W#16#0;
   STAT01[84] := W#16#0;
   STAT01[85] := W#16#0;
   STAT01[86] := W#16#0;
   STAT01[87] := W#16#0;
   STAT01[88] := W#16#0;
   STAT01[89] := W#16#0;
   STAT01[90] := W#16#0;
   STAT01[91] := W#16#0;
   STAT01[92] := W#16#0;
   STAT01[93] := W#16#0;
   STAT01[94] := W#16#0;
   STAT01[95] := W#16#0;
   STAT01[96] := W#16#0;
   STAT01[97] := W#16#0;
   STAT01[98] := W#16#0;
   STAT01[99] := W#16#0;
   STAT011[0] := W#16#0;
   STAT011[1] := W#16#0;
   STAT011[2] := W#16#0;
   STAT011[3] := W#16#0;
   STAT011[4] := W#16#0;
   STAT011[5] := W#16#0;
   STAT011[6] := W#16#0;
   STAT011[7] := W#16#0;
   STAT011[8] := W#16#0;
   STAT011[9] := W#16#0;
   STAT011[10] := W#16#0;
   STAT011[11] := W#16#0;
   STAT011[12] := W#16#0;
   STAT011[13] := W#16#0;
   STAT011[14] := W#16#0;
   STAT011[15] := W#16#0;
   STAT011[16] := W#16#0;
   STAT011[17] := W#16#0;
   STAT011[18] := W#16#0;
   STAT011[19] := W#16#0;
   STAT011[20] := W#16#0;
   STAT011[21] := W#16#0;
   STAT011[22] := W#16#0;
   STAT011[23] := W#16#0;
   STAT011[24] := W#16#0;
   STAT011[25] := W#16#0;
   STAT011[26] := W#16#0;
   STAT011[27] := W#16#0;
   STAT011[28] := W#16#0;
   STAT011[29] := W#16#0;
   STAT011[30] := W#16#0;
   STAT011[31] := W#16#0;
   STAT011[32] := W#16#0;
   STAT011[33] := W#16#0;
   STAT011[34] := W#16#0;
   STAT011[35] := W#16#0;
   STAT011[36] := W#16#0;
   STAT011[37] := W#16#0;
   STAT011[38] := W#16#0;
   STAT011[39] := W#16#0;
   STAT011[40] := W#16#0;
   STAT011[41] := W#16#0;
   STAT011[42] := W#16#0;
   STAT011[43] := W#16#0;
   STAT011[44] := W#16#0;
   STAT011[45] := W#16#0;
   STAT011[46] := W#16#0;
   STAT011[47] := W#16#0;
   STAT011[48] := W#16#0;
   STAT011[49] := W#16#0;
   STAT011[50] := W#16#0;
   STAT011[51] := W#16#0;
   STAT011[52] := W#16#0;
   STAT011[53] := W#16#0;
   STAT011[54] := W#16#0;
   STAT011[55] := W#16#0;
   STAT011[56] := W#16#0;
   STAT011[57] := W#16#0;
   STAT011[58] := W#16#0;
   STAT011[59] := W#16#0;
   STAT011[60] := W#16#0;
   STAT011[61] := W#16#0;
   STAT011[62] := W#16#0;
   STAT011[63] := W#16#0;
   STAT011[64] := W#16#0;
   STAT011[65] := W#16#0;
   STAT011[66] := W#16#0;
   STAT011[67] := W#16#0;
   STAT011[68] := W#16#0;
   STAT011[69] := W#16#0;
   STAT011[70] := W#16#0;
   STAT011[71] := W#16#0;
   STAT011[72] := W#16#0;
   STAT011[73] := W#16#0;
   STAT011[74] := W#16#0;
   STAT011[75] := W#16#0;
   STAT011[76] := W#16#0;
   STAT011[77] := W#16#0;
   STAT011[78] := W#16#0;
   STAT011[79] := W#16#0;
   STAT011[80] := W#16#0;
   STAT011[81] := W#16#0;
   STAT011[82] := W#16#0;
   STAT011[83] := W#16#0;
   STAT011[84] := W#16#0;
   STAT011[85] := W#16#0;
   STAT011[86] := W#16#0;
   STAT011[87] := W#16#0;
   STAT011[88] := W#16#0;
   STAT011[89] := W#16#0;
   STAT011[90] := W#16#0;
   STAT011[91] := W#16#0;
   STAT011[92] := W#16#0;
   STAT011[93] := W#16#0;
   STAT011[94] := W#16#0;
   STAT011[95] := W#16#0;
   STAT011[96] := W#16#0;
   STAT011[97] := W#16#0;
   STAT011[98] := W#16#0;
   STAT011[99] := W#16#0;
END_DATA_BLOCK

DATA_BLOCK DB 51
TITLE =
VERSION : 0.1


  STRUCT
   S_SHUTTLE : STRUCT
    M_AUTO_SEL : BOOL ;
    M_MANUAL_SEL : BOOL ;
    M_READY_PB : BOOL ;
    M_AUTO_RUN_PB : BOOL ;
    M_WORK_COMP_SET_PB : BOOL ;
    M_WORK_COMP_RST_PB : BOOL ;
    M_HOME_POS_PB : BOOL ;
    M_TIP_DRESS_PB : BOOL ;
    HOOK_PIN_SEL : BOOL ;
    DAECHA_LOCK_SEL : BOOL ;
    ELE_SEL : BOOL ;
    AIR_ELE_SEL : BOOL ;
    SPARE13 : BOOL ;
    SPARE14 : BOOL ;
    SPARE15 : BOOL ;
    M_ALL_TIP_DRESS_PB : BOOL ;
    SPARE17 : BOOL ;
    SPARE18 : BOOL ;
    SPARE19 : BOOL ;
    SPARE20 : BOOL ;
    SPARE21 : BOOL ;
    SPARE22 : BOOL ;
    SPARE23 : BOOL ;
    SPARE24 : BOOL ;
    SERVO_LOW_SS : BOOL ;
    SERVO_HIGH_SS : BOOL ;
    MELODY_ON_PB : BOOL ;
    SPARE28 : BOOL ;
    SPARE29 : BOOL ;
    SPARE30 : BOOL ;
    M_ADV_PB : BOOL ;
    M_RET_PB : BOOL ;
    SPARE33 : BOOL ;
    SPARE34 : BOOL ;
    SPARE35 : BOOL ;
    SPARE36 : BOOL ;
    SPARE37 : BOOL ;
    SPARE38 : BOOL ;
    SPARE39 : BOOL ;
    SPARE40 : BOOL ;
    SPARE41 : BOOL ;
    SPARE42 : BOOL ;
    SPARE43 : BOOL ;
    SPARE44 : BOOL ;
    SPARE45 : BOOL ;
    SPARE46 : BOOL ;
    SPARE47 : BOOL ;
    SPARE48 : BOOL ;
    SPARE50 : BOOL ;
    SPARE51 : BOOL ;
    SPARE52 : BOOL ;
    SPARE53 : BOOL ;
    SPARE54 : BOOL ;
    SPARE55 : BOOL ;
    SPARE56 : BOOL ;
    SPARE57 : BOOL ;
    SPARE58 : BOOL ;
    SPARE59 : BOOL ;
    SPARE60 : BOOL ;
    SPARE61 : BOOL ;
    SPARE62 : BOOL ;
    SPARE63 : BOOL ;
    SPARE64 : BOOL ;
    SPARE65 : BOOL ;
    SPARE66 : BOOL ;
    SPARE67 : BOOL ;
    SPARE68 : BOOL ;
    SPARE69 : BOOL ;
    SPARE70 : BOOL ;
    SPARE71 : BOOL ;
    SPARE72 : BOOL ;
    SPARE73 : BOOL ;
    SPARE74 : BOOL ;
    SPARE75 : BOOL ;
    SPARE76 : BOOL ;
    SPARE77 : BOOL ;
    SPARE78 : BOOL ;
    SPARE79 : BOOL ;
    SPARE80 : BOOL ;
    SPARE81 : BOOL ;
    SPARE82 : BOOL ;
    SPARE83 : BOOL ;
    SPARE84 : BOOL ;
    SPARE85 : BOOL ;
    SPARE86 : BOOL ;
    SPARE87 : BOOL ;
    SPARE88 : BOOL ;
    SPARE89 : BOOL ;
    SPARE90 : BOOL ;
    SPARE91 : BOOL ;
    SPARE92 : BOOL ;
    SPARE93 : BOOL ;
    SPARE94 : BOOL ;
    SPARE95 : BOOL ;
    SPARE96 : BOOL ;
    SPARE97 : BOOL ;
    SPARE98 : BOOL ;
    SPARE99 : BOOL ;
    SPARE100 : BOOL ;
    SPARE101 : BOOL ;
    SPARE102 : BOOL ;
    SPARE103 : BOOL ;
    SPARE104 : BOOL ;
    SPARE105 : BOOL ;
    SPARE106 : BOOL ;
    SPARE107 : BOOL ;
    SPARE108 : BOOL ;
    SPARE109 : BOOL ;
    SPARE110 : BOOL ;
    SPARE111 : BOOL ;
    SPARE112 : BOOL ;
    SPARE113 : BOOL ;
    SPARE114 : BOOL ;
    SPARE115 : BOOL ;
    SPARE116 : BOOL ;
    SPARE117 : BOOL ;
    SPARE118 : BOOL ;
    SPARE119 : BOOL ;
    SPARE120 : BOOL ;
    SPARE121 : BOOL ;
    SPARE122 : BOOL ;
    SPARE123 : BOOL ;
    SPARE124 : BOOL ;
    SPARE125 : BOOL ;
    SPARE126 : BOOL ;
    SPARE127 : BOOL ;
    SPARE128 : BOOL ;
    SPARE129 : BOOL ;
    SPARE130 : BOOL ;
    SPARE131 : BOOL ;
    SPARE132 : BOOL ;
    SPARE133 : BOOL ;
    SPARE134 : BOOL ;
    SPARE135 : BOOL ;
    SPARE136 : BOOL ;
    SPARE137 : BOOL ;
    SPARE138 : BOOL ;
    SPARE139 : BOOL ;
    SPARE140 : BOOL ;
    SPARE141 : BOOL ;
    SPARE142 : BOOL ;
    SPARE143 : BOOL ;
    SPARE144 : BOOL ;
    SPARE145 : BOOL ;
    SPARE146 : BOOL ;
    SPARE147 : BOOL ;
    SPARE148 : BOOL ;
    SPARE149 : BOOL ;
    SPARE150 : BOOL ;
    SPARE151 : BOOL ;
    SPARE152 : BOOL ;
    SPARE153 : BOOL ;
    SPARE154 : BOOL ;
    SPARE155 : BOOL ;
    SPARE156 : BOOL ;
    SPARE157 : BOOL ;
    SPARE158 : BOOL ;
    SPARE159 : BOOL ;
    SPARE160 : BOOL ;
    SPARE161 : BOOL ;
    HOOK_PIN_UP_LP : WORD ;
    HOOK_PIN_DOWN_LP : WORD ;
    DAECHA_LOCK_ADV_LP : WORD ;
    DAECHA_LOCK_RET_LP : WORD ;
    ELE_ADV_LP : WORD ;
    ELE_RET_LP : WORD ;
    AIR_ELE_ADV_LP : WORD ;
    AIR_ELE_RET_LP : WORD ;
    SP_WORD19 : WORD ;
    SP_WORD20 : WORD ;
    LM_DC_PIN_UP_LP : WORD ;
    LM_DC_PIN_DOWN_LP : WORD ;
    LM_DC_1ST_CLAMP1_ADV_LP : WORD ;
    LM_DC_1ST_CLAMP1_RET_LP : WORD ;
    LM_DC_1ST_CLAMP2_ADV_LP : WORD ;
    LM_DC_1ST_CLAMP2_RET_LP : WORD ;
    LM_DC_1ST_CLAMP3_ADV_LP : WORD ;
    LM_DC_1ST_CLAMP3_RET_LP : WORD ;
    LM_DC_1ST_CLAMP4_ADV_LP : WORD ;
    LM_DC_1ST_CLAMP4_RET_LP : WORD ;
    LM_DC_2ND_CLAMP1_ADV_LP : WORD ;
    LM_DC_2ND_CLAMP1_RET_LP : WORD ;
    LM_DC_2ND_CLAMP2_ADV_LP : WORD ;
    LM_DC_2ND_CLAMP2_RET_LP : WORD ;
    LM_DC_2ND_CLAMP3_ADV_LP : WORD ;
    LM_DC_2ND_CLAMP3_RET_LP : WORD ;
    LM_DC_2ND_CLAMP4_ADV_LP : WORD ;
    LM_DC_2ND_CLAMP4_RET_LP : WORD ;
    LM_DC_2ND_CLAMP5_ADV_LP : WORD ;
    LM_DC_2ND_CLAMP5_RET_LP : WORD ;
    LM_DC_DR_STK_PIN_UP_LP : WORD ;
    LM_DC_DR_STK_PIN_DOWN_LP : WORD ;
    LM_DC_OTR_CLAMP_ADV_LP : WORD ;
    LM_DC_OTR_CLAMP_RET_LP : WORD ;
    LM_DC_ASSY_CLAMP_ADV_LP : WORD ;
    LM_DC_ASSY_CLAMP_RET_LP : WORD ;
    LM_DC_FF_PIN_UP_LP : WORD ;
    LM_DC_FF_PIN_DOWN_LP : WORD ;
    LM_DC_FF_CLAMP_ADV_LP : WORD ;
    LM_DC_FF_CLAMP_RET_LP : WORD ;
    LM_DC_2ND_CLAMP6_ADV_LP : WORD ;
    LM_DC_2ND_CLAMP6_RET_LP : WORD ;
    LM_DC_2ND_CLAMP7_ADV_LP : WORD ;
    LM_DC_2ND_CLAMP7_RET_LP : WORD ;
    LM_DC_1ST_CLAMP5_ADV_LP : WORD ;
    LM_DC_1ST_CLAMP5_RET_LP : WORD ;
    SP_WORD68 : WORD ;
    SP_WORD69 : WORD ;
    SP_WORD70 : WORD ;
    SP_WORD71 : WORD ;
    TL_DC_PIN_UP_LP : WORD ;
    TL_DC_PIN_DOWN_LP : WORD ;
    TL_DC_LATCH1_ADV_LP : WORD ;
    TL_DC_LATCH1_RET_LP : WORD ;
    TL_DC_LATCH2_ADV_LP : WORD ;
    TL_DC_LATCH2_RET_LP : WORD ;
    TL_DC_1ST_CLAMP1_ADV_LP : WORD ;
    TL_DC_1ST_CLAMP1_RET_LP : WORD ;
    TL_DC_1ST_CLAMP2_ADV_LP : WORD ;
    TL_DC_1ST_CLAMP2_RET_LP : WORD ;
    TL_DC_1ST_CLAMP3_ADV_LP : WORD ;
    TL_DC_1ST_CLAMP3_RET_LP : WORD ;
    TL_DC_2ND_CLAMP1_ADV_LP : WORD ;
    TL_DC_2ND_CLAMP1_RET_LP : WORD ;
    TL_DC_2ND_CLAMP2_ADV_LP : WORD ;
    TL_DC_2ND_CLAMP2_RET_LP : WORD ;
    TL_DC_U261_ADV_LP : WORD ;
    TL_DC_U261_RET_LP : WORD ;
    TL_DC_U261_CLAMP_ADV_LP : WORD ;
    TL_DC_U261_CLAMP_RET_LP : WORD ;
    TL_DC_U269_UP_LP : WORD ;
    TL_DC_U269_DOWN_LP : WORD ;
    TL_DC_U269_CLAMP_ADV_LP : WORD ;
    TL_DC_U269_CLAMP_RET_LP : WORD ;
    TL_DC_3RD_CLAMP_ADV_LP : WORD ;
    TL_DC_3RD_CLAMP_RET_LP : WORD ;
    TL_DC_U262_1_UP_LP : WORD ;
    TL_DC_U262_1_DOWN_LP : WORD ;
    TL_DC_U262_1_ADV_LP : WORD ;
    TL_DC_U262_1_RET_LP : WORD ;
    TL_DC_U262_1_CLP_ADV_LP : WORD ;
    TL_DC_U262_1_CLP_RET_LP : WORD ;
    TL_DC_U261_2_CLP_ADV_LP : WORD ;
    TL_DC_U261_2_CLP_RET_LP : WORD ;
    SP_WORD106 : WORD ;
    SP_WORD107 : WORD ;
    SP_WORD108 : WORD ;
    SP_WORD109 : WORD ;
    SP_WORD110 : WORD ;
    SP_WORD111 : WORD ;
   END_STRUCT ;
   S_702 : STRUCT
    M_AUTO_SEL : BOOL ;
    M_MANUAL_SEL : BOOL ;
    M_READY_PB : BOOL ;
    M_AUTO_RUN_PB : BOOL ;
    M_WORK_COMP_SET_PB : BOOL ;
    M_WORK_COMP_RST_PB : BOOL ;
    M_HOME_POS_PB : BOOL ;
    M_TIP_DRESS_PB : BOOL ;
    HOOK_PIN_SEL : BOOL ;
    DAECHA_LOCK_SEL : BOOL ;
    DAECHA_LOCK_UP_DN_SEL : BOOL ;
    AIR_ELE_SEL : BOOL ;
    EJECT_SEL : BOOL ;
    STOPPER_SER : BOOL ;
    DAECHA_CLAMP_SEL : BOOL ;
    SHOCK_ABSORBER_SEL : BOOL ;
    DAECHA_IN_SEL : BOOL ;
    DAECHA_OUT_SEL : BOOL ;
    SPARE19 : BOOL ;
    SPARE20 : BOOL ;
    SPARE21 : BOOL ;
    SPARE22 : BOOL ;
    SPARE23 : BOOL ;
    SPARE24 : BOOL ;
    LINE_EMPTY_SS : BOOL ;
    OUT_TRV_BT_ON_PB : BOOL ;
    SPARE27 : BOOL ;
    SPARE28 : BOOL ;
    SPARE29 : BOOL ;
    SPARE30 : BOOL ;
    M_ADV_PB : BOOL ;
    M_RET_PB : BOOL ;
    LM_DC_PIN_SEL : BOOL ;
    LM_DC_1ST_CLAMP1_SEL : BOOL ;
    LM_DC_1ST_CLAMP2_SEL : BOOL ;
    LM_DC_1ST_CLAMP3_SEL : BOOL ;
    LM_DC_1ST_CLAMP4_SEL : BOOL ;
    LM_DC_2ND_CLAMP1_SEL : BOOL ;
    LM_DC_2ND_CLAMP2_SEL : BOOL ;
    LM_DC_2ND_CLAMP3_SEL : BOOL ;
    LM_DC_2ND_CLAMP4_SEL : BOOL ;
    LM_DC_2ND_CLAMP5_SEL : BOOL ;
    LM_DC_DR_STK_PIN_SEL : BOOL ;
    LM_DC_OTR_CLAMP_SEL : BOOL ;
    LM_DC_ASSY_CLAMP_SEL : BOOL ;
    LM_DC_FF_PIN_SEL : BOOL ;
    LM_DC_FF_CLAMP_SEL : BOOL ;
    LM_DC_2ND_CLAMP6_SEL : BOOL ;
    SPARE50 : BOOL ;
    SPARE51 : BOOL ;
    SPARE52 : BOOL ;
    SPARE53 : BOOL ;
    SPARE54 : BOOL ;
    SPARE55 : BOOL ;
    SPARE56 : BOOL ;
    SPARE57 : BOOL ;
    SPARE58 : BOOL ;
    SPARE59 : BOOL ;
    SPARE60 : BOOL ;
    SPARE61 : BOOL ;
    SPARE62 : BOOL ;
    SPARE63 : BOOL ;
    LM_DC_M_ADV_PB : BOOL ;
    LM_DC_M_RET_PB : BOOL ;
    TL_DC_PIN_SEL : BOOL ;
    TL_DC_LATCH1_SEL : BOOL ;
    TL_DC_1ST_CLAMP_SEL : BOOL ;
    TL_DC_2ND_CLAMP_SEL : BOOL ;
    TL_DC_U261_SEL : BOOL ;
    TL_DC_U261_CLAMP_SEL : BOOL ;
    TL_DC_U269_UP_DN_SEL : BOOL ;
    TL_DC_U269_CLAMP_SEL : BOOL ;
    TL_DC_3RD_CLAMP_SEL : BOOL ;
    TL_DC_U262_1_UP_DN_SEL : BOOL ;
    TL_DC_U262_1_SEL : BOOL ;
    TL_DC_U262_1_CLAMP_SEL : BOOL ;
    TL_DC_U261_2_CLAMP_SEL : BOOL ;
    SPARE79 : BOOL ;
    SPARE80 : BOOL ;
    SPARE81 : BOOL ;
    SPARE82 : BOOL ;
    SPARE83 : BOOL ;
    SPARE84 : BOOL ;
    SPARE85 : BOOL ;
    SPARE86 : BOOL ;
    SPARE87 : BOOL ;
    SPARE88 : BOOL ;
    SPARE89 : BOOL ;
    SPARE90 : BOOL ;
    SPARE91 : BOOL ;
    SPARE92 : BOOL ;
    SPARE93 : BOOL ;
    SPARE94 : BOOL ;
    SPARE95 : BOOL ;
    TL_DC_M_ADV_PB : BOOL ;
    TL_DC_M_RET_PB : BOOL ;
    SPARE98 : BOOL ;
    SPARE99 : BOOL ;
    SPARE100 : BOOL ;
    SPARE101 : BOOL ;
    SPARE102 : BOOL ;
    SPARE103 : BOOL ;
    SPARE104 : BOOL ;
    SPARE105 : BOOL ;
    SPARE106 : BOOL ;
    SPARE107 : BOOL ;
    SPARE108 : BOOL ;
    SPARE109 : BOOL ;
    SPARE110 : BOOL ;
    SPARE111 : BOOL ;
    SPARE112 : BOOL ;
    SPARE113 : BOOL ;
    SPARE114 : BOOL ;
    SPARE115 : BOOL ;
    SPARE116 : BOOL ;
    SPARE117 : BOOL ;
    SPARE118 : BOOL ;
    SPARE119 : BOOL ;
    SPARE120 : BOOL ;
    SPARE121 : BOOL ;
    SPARE122 : BOOL ;
    SPARE123 : BOOL ;
    SPARE124 : BOOL ;
    SPARE125 : BOOL ;
    SPARE126 : BOOL ;
    SPARE127 : BOOL ;
    SPARE128 : BOOL ;
    SPARE129 : BOOL ;
    SPARE130 : BOOL ;
    SPARE131 : BOOL ;
    SPARE132 : BOOL ;
    SPARE133 : BOOL ;
    SPARE134 : BOOL ;
    SPARE135 : BOOL ;
    SPARE136 : BOOL ;
    SPARE137 : BOOL ;
    SPARE138 : BOOL ;
    SPARE139 : BOOL ;
    SPARE140 : BOOL ;
    SPARE141 : BOOL ;
    SPARE142 : BOOL ;
    SPARE143 : BOOL ;
    SPARE144 : BOOL ;
    SPARE145 : BOOL ;
    SPARE146 : BOOL ;
    SPARE147 : BOOL ;
    SPARE148 : BOOL ;
    SPARE149 : BOOL ;
    SPARE150 : BOOL ;
    SPARE151 : BOOL ;
    SPARE152 : BOOL ;
    SPARE153 : BOOL ;
    SPARE154 : BOOL ;
    SPARE155 : BOOL ;
    SPARE156 : BOOL ;
    SPARE157 : BOOL ;
    SPARE158 : BOOL ;
    SPARE159 : BOOL ;
    SPARE160 : BOOL ;
    SPARE161 : BOOL ;
    HOOK_PIN_UP_LP : WORD ;
    HOOK_PIN_DOWN_LP : WORD ;
    DAECHA_LOCK_ADV_LP : WORD ;
    DAECHA_LOCK_RET_LP : WORD ;
    DAECHA_LOCK_UP_LP : WORD ;
    DAECHA_LOCK_DOWN_LP : WORD ;
    ELE_ADV_LP : WORD ;
    ELE_RET_LP : WORD ;
    AIR_ELE_ADV_LP : WORD ;
    AIR_ELE_RET_LP : WORD ;
    LM_DC_PIN_UP_LP : WORD ;
    LM_DC_PIN_DOWN_LP : WORD ;
    LM_DC_1ST_CLAMP1_ADV_LP : WORD ;
    LM_DC_1ST_CLAMP1_RET_LP : WORD ;
    LM_DC_1ST_CLAMP2_ADV_LP : WORD ;
    LM_DC_1ST_CLAMP2_RET_LP : WORD ;
    LM_DC_1ST_CLAMP3_ADV_LP : WORD ;
    LM_DC_1ST_CLAMP3_RET_LP : WORD ;
    LM_DC_1ST_CLAMP4_ADV_LP : WORD ;
    LM_DC_1ST_CLAMP4_RET_LP : WORD ;
    LM_DC_2ND_CLAMP1_ADV_LP : WORD ;
    LM_DC_2ND_CLAMP1_RET_LP : WORD ;
    LM_DC_2ND_CLAMP2_ADV_LP : WORD ;
    LM_DC_2ND_CLAMP2_RET_LP : WORD ;
    LM_DC_2ND_CLAMP3_ADV_LP : WORD ;
    LM_DC_2ND_CLAMP3_RET_LP : WORD ;
    LM_DC_2ND_CLAMP4_ADV_LP : WORD ;
    LM_DC_2ND_CLAMP4_RET_LP : WORD ;
    LM_DC_2ND_CLAMP5_ADV_LP : WORD ;
    LM_DC_2ND_CLAMP5_RET_LP : WORD ;
    LM_DC_DR_STK_PIN_UP_LP : WORD ;
    LM_DC_DR_STK_PIN_DOWN_LP : WORD ;
    LM_DC_OTR_CLAMP_ADV_LP : WORD ;
    LM_DC_OTR_CLAMP_RET_LP : WORD ;
    LM_DC_ASSY_CLAMP_ADV_LP : WORD ;
    LM_DC_ASSY_CLAMP_RET_LP : WORD ;
    LM_DC_FF_PIN_UP_LP : WORD ;
    LM_DC_FF_PIN_DOWN_LP : WORD ;
    LM_DC_FF_CLAMP_ADV_LP : WORD ;
    LM_DC_FF_CLAMP_RET_LP : WORD ;
    LM_DC_2ND_CLAMP6_ADV_LP : WORD ;
    LM_DC_2ND_CLAMP6_RET_LP : WORD ;
    LM_DC_2ND_CLAMP7_ADV_LP : WORD ;
    LM_DC_2ND_CLAMP7_RET_LP : WORD ;
    LM_DC_1ST_CLAMP5_ADV_LP : WORD ;
    LM_DC_1ST_CLAMP5_RET_LP : WORD ;
    EJECT_UP_LP : WORD ;
    EJECT_DOWN_LP : WORD ;
    STOPPER_ADV_LP : WORD ;
    STOPPER_RET_LP : WORD ;
    TL_DC_PIN_UP_LP : WORD ;
    TL_DC_PIN_DOWN_LP : WORD ;
    TL_DC_LATCH1_ADV_LP : WORD ;
    TL_DC_LATCH1_RET_LP : WORD ;
    TL_DC_LATCH2_ADV_LP : WORD ;
    TL_DC_LATCH2_RET_LP : WORD ;
    TL_DC_1ST_CLAMP1_ADV_LP : WORD ;
    TL_DC_1ST_CLAMP1_RET_LP : WORD ;
    TL_DC_1ST_CLAMP2_ADV_LP : WORD ;
    TL_DC_1ST_CLAMP2_RET_LP : WORD ;
    TL_DC_1ST_CLAMP3_ADV_LP : WORD ;
    TL_DC_1ST_CLAMP3_RET_LP : WORD ;
    TL_DC_2ND_CLAMP1_ADV_LP : WORD ;
    TL_DC_2ND_CLAMP1_RET_LP : WORD ;
    TL_DC_2ND_CLAMP2_ADV_LP : WORD ;
    TL_DC_2ND_CLAMP2_RET_LP : WORD ;
    TL_DC_U261_ADV_LP : WORD ;
    TL_DC_U261_RET_LP : WORD ;
    TL_DC_U261_CLAMP_ADV_LP : WORD ;
    TL_DC_U261_CLAMP_RET_LP : WORD ;
    TL_DC_U269_UP_LP : WORD ;
    TL_DC_U269_DOWN_LP : WORD ;
    TL_DC_U269_CLAMP_ADV_LP : WORD ;
    TL_DC_U269_CLAMP_RET_LP : WORD ;
    TL_DC_3RD_CLAMP_ADV_LP : WORD ;
    TL_DC_3RD_CLAMP_RET_LP : WORD ;
    TL_DC_U262_1_UP_LP : WORD ;
    TL_DC_U262_1_DOWN_LP : WORD ;
    TL_DC_U262_1_ADV_LP : WORD ;
    TL_DC_U262_1_RET_LP : WORD ;
    TL_DC_U262_1_CLP_ADV_LP : WORD ;
    TL_DC_U262_1_CLP_RET_LP : WORD ;
    TL_DC_U261_2_CLP_ADV_LP : WORD ;
    TL_DC_U261_2_CLP_RET_LP : WORD ;
    SP_WORD106 : WORD ;
    SP_WORD107 : WORD ;
    DAECHA_CLAMP_ADV_LP : WORD ;
    DAECHA_CLAMP_RET_LP : WORD ;
    SHOCK_ABSORBER_ADV_LP : WORD ;
    SHOCK_ABSORBER_RET_LP : WORD ;
   END_STRUCT ;
   S_703 : STRUCT
    M_AUTO_SEL : BOOL ;
    M_MANUAL_SEL : BOOL ;
    M_READY_PB : BOOL ;
    M_AUTO_RUN_PB : BOOL ;
    M_WORK_COMP_SET_PB : BOOL ;
    M_WORK_COMP_RST_PB : BOOL ;
    M_HOME_POS_PB : BOOL ;
    M_TIP_DRESS_PB : BOOL ;
    HOOK_PIN_SEL : BOOL ;
    DAECHA_LOCK_SEL : BOOL ;
    ELE_SEL : BOOL ;
    SPARE12 : BOOL ;
    SPARE13 : BOOL ;
    SPARE14 : BOOL ;
    SPARE15 : BOOL ;
    SPARE16 : BOOL ;
    SPARE17 : BOOL ;
    SPARE18 : BOOL ;
    SPARE19 : BOOL ;
    SPARE20 : BOOL ;
    SPARE21 : BOOL ;
    SPARE22 : BOOL ;
    SPARE23 : BOOL ;
    SPARE24 : BOOL ;
    SPARE25 : BOOL ;
    SPARE26 : BOOL ;
    SPARE27 : BOOL ;
    SPARE28 : BOOL ;
    SPARE29 : BOOL ;
    SPARE30 : BOOL ;
    M_ADV_PB : BOOL ;
    M_RET_PB : BOOL ;
    LM_DC_PIN_SEL : BOOL ;
    LM_DC_1ST_CLAMP1_SEL : BOOL ;
    LM_DC_1ST_CLAMP2_SEL : BOOL ;
    LM_DC_1ST_CLAMP3_SEL : BOOL ;
    LM_DC_1ST_CLAMP4_SEL : BOOL ;
    LM_DC_2ND_CLAMP1_SEL : BOOL ;
    LM_DC_2ND_CLAMP2_SEL : BOOL ;
    LM_DC_2ND_CLAMP3_SEL : BOOL ;
    LM_DC_2ND_CLAMP4_SEL : BOOL ;
    LM_DC_2ND_CLAMP5_SEL : BOOL ;
    LM_DC_DR_STK_PIN_SEL : BOOL ;
    LM_DC_OTR_CLAMP_SEL : BOOL ;
    LM_DC_ASSY_CLAMP_SEL : BOOL ;
    LM_DC_FF_PIN_SEL : BOOL ;
    LM_DC_FF_CLAMP_SEL : BOOL ;
    LM_DC_2ND_CLAMP6_SEL : BOOL ;
    SPARE50 : BOOL ;
    SPARE51 : BOOL ;
    SPARE52 : BOOL ;
    SPARE53 : BOOL ;
    SPARE54 : BOOL ;
    SPARE55 : BOOL ;
    SPARE56 : BOOL ;
    SPARE57 : BOOL ;
    SPARE58 : BOOL ;
    SPARE59 : BOOL ;
    SPARE60 : BOOL ;
    SPARE61 : BOOL ;
    SPARE62 : BOOL ;
    SPARE63 : BOOL ;
    LM_DC_M_ADV_PB : BOOL ;
    LM_DC_M_RET_PB : BOOL ;
    TL_DC_PIN_SEL : BOOL ;
    TL_DC_LATCH1_SEL : BOOL ;
    TL_DC_1ST_CLAMP_SEL : BOOL ;
    TL_DC_2ND_CLAMP_SEL : BOOL ;
    TL_DC_U261_SEL : BOOL ;
    TL_DC_U261_CLAMP_SEL : BOOL ;
    TL_DC_U269_UP_DN_SEL : BOOL ;
    TL_DC_U269_CLAMP_SEL : BOOL ;
    TL_DC_3RD_CLAMP_SEL : BOOL ;
    TL_DC_U262_1_UP_DN_SEL : BOOL ;
    TL_DC_U262_1_SEL : BOOL ;
    TL_DC_U262_1_CLAMP_SEL : BOOL ;
    TL_DC_U261_2_CLAMP_SEL : BOOL ;
    SPARE79 : BOOL ;
    SPARE80 : BOOL ;
    SPARE81 : BOOL ;
    SPARE82 : BOOL ;
    SPARE83 : BOOL ;
    SPARE84 : BOOL ;
    SPARE85 : BOOL ;
    SPARE86 : BOOL ;
    SPARE87 : BOOL ;
    SPARE88 : BOOL ;
    SPARE89 : BOOL ;
    SPARE90 : BOOL ;
    SPARE91 : BOOL ;
    SPARE92 : BOOL ;
    SPARE93 : BOOL ;
    SPARE94 : BOOL ;
    SPARE95 : BOOL ;
    TL_DC_M_ADV_PB : BOOL ;
    TL_DC_M_RET_PB : BOOL ;
    SPARE98 : BOOL ;
    SPARE99 : BOOL ;
    SPARE100 : BOOL ;
    SPARE101 : BOOL ;
    SPARE102 : BOOL ;
    SPARE103 : BOOL ;
    SPARE104 : BOOL ;
    SPARE105 : BOOL ;
    SPARE106 : BOOL ;
    SPARE107 : BOOL ;
    SPARE108 : BOOL ;
    SPARE109 : BOOL ;
    SPARE110 : BOOL ;
    SPARE111 : BOOL ;
    SPARE112 : BOOL ;
    SPARE113 : BOOL ;
    SPARE114 : BOOL ;
    SPARE115 : BOOL ;
    SPARE116 : BOOL ;
    SPARE117 : BOOL ;
    SPARE118 : BOOL ;
    SPARE119 : BOOL ;
    SPARE120 : BOOL ;
    SPARE121 : BOOL ;
    SPARE122 : BOOL ;
    SPARE123 : BOOL ;
    SPARE124 : BOOL ;
    SPARE125 : BOOL ;
    SPARE126 : BOOL ;
    SPARE127 : BOOL ;
    SPARE128 : BOOL ;
    SPARE129 : BOOL ;
    SPARE130 : BOOL ;
    SPARE131 : BOOL ;
    SPARE132 : BOOL ;
    SPARE133 : BOOL ;
    SPARE134 : BOOL ;
    SPARE135 : BOOL ;
    SPARE136 : BOOL ;
    SPARE137 : BOOL ;
    SPARE138 : BOOL ;
    SPARE139 : BOOL ;
    SPARE140 : BOOL ;
    SPARE141 : BOOL ;
    SPARE142 : BOOL ;
    SPARE143 : BOOL ;
    SPARE144 : BOOL ;
    SPARE145 : BOOL ;
    SPARE146 : BOOL ;
    SPARE147 : BOOL ;
    SPARE148 : BOOL ;
    SPARE149 : BOOL ;
    SPARE150 : BOOL ;
    SPARE151 : BOOL ;
    SPARE152 : BOOL ;
    SPARE153 : BOOL ;
    SPARE154 : BOOL ;
    SPARE155 : BOOL ;
    SPARE156 : BOOL ;
    SPARE157 : BOOL ;
    SPARE158 : BOOL ;
    SPARE159 : BOOL ;
    SPARE160 : BOOL ;
    SPARE161 : BOOL ;
    HOOK_PIN_UP_LP : WORD ;
    HOOK_PIN_DOWN_LP : WORD ;
    DAECHA_LOCK_ADV_LP : WORD ;
    DAECHA_LOCK_RET_LP : WORD ;
    ELE_ADV_LP : WORD ;
    ELE_RET_LP : WORD ;
    AIR_ELE_ADV_LP : WORD ;
    AIR_ELE_RET_LP : WORD ;
    SP_WORD19 : WORD ;
    SP_WORD20 : WORD ;
    LM_DC_PIN_UP_LP : WORD ;
    LM_DC_PIN_DOWN_LP : WORD ;
    LM_DC_1ST_CLAMP1_ADV_LP : WORD ;
    LM_DC_1ST_CLAMP1_RET_LP : WORD ;
    LM_DC_1ST_CLAMP2_ADV_LP : WORD ;
    LM_DC_1ST_CLAMP2_RET_LP : WORD ;
    LM_DC_1ST_CLAMP3_ADV_LP : WORD ;
    LM_DC_1ST_CLAMP3_RET_LP : WORD ;
    LM_DC_1ST_CLAMP4_ADV_LP : WORD ;
    LM_DC_1ST_CLAMP4_RET_LP : WORD ;
    LM_DC_2ND_CLAMP1_ADV_LP : WORD ;
    LM_DC_2ND_CLAMP1_RET_LP : WORD ;
    LM_DC_2ND_CLAMP2_ADV_LP : WORD ;
    LM_DC_2ND_CLAMP2_RET_LP : WORD ;
    LM_DC_2ND_CLAMP3_ADV_LP : WORD ;
    LM_DC_2ND_CLAMP3_RET_LP : WORD ;
    LM_DC_2ND_CLAMP4_ADV_LP : WORD ;
    LM_DC_2ND_CLAMP4_RET_LP : WORD ;
    LM_DC_2ND_CLAMP5_ADV_LP : WORD ;
    LM_DC_2ND_CLAMP5_RET_LP : WORD ;
    LM_DC_DR_STK_PIN_UP_LP : WORD ;
    LM_DC_DR_STK_PIN_DOWN_LP : WORD ;
    LM_DC_OTR_CLAMP_ADV_LP : WORD ;
    LM_DC_OTR_CLAMP_RET_LP : WORD ;
    LM_DC_ASSY_CLAMP_ADV_LP : WORD ;
    LM_DC_ASSY_CLAMP_RET_LP : WORD ;
    LM_DC_FF_PIN_UP_LP : WORD ;
    LM_DC_FF_PIN_DOWN_LP : WORD ;
    LM_DC_FF_CLAMP_ADV_LP : WORD ;
    LM_DC_FF_CLAMP_RET_LP : WORD ;
    LM_DC_2ND_CLAMP6_ADV_LP : WORD ;
    LM_DC_2ND_CLAMP6_RET_LP : WORD ;
    LM_DC_2ND_CLAMP7_ADV_LP : WORD ;
    LM_DC_2ND_CLAMP7_RET_LP : WORD ;
    LM_DC_1ST_CLAMP5_ADV_LP : WORD ;
    LM_DC_1ST_CLAMP5_RET_LP : WORD ;
    SP_WORD68 : WORD ;
    SP_WORD69 : WORD ;
    SP_WORD70 : WORD ;
    SP_WORD71 : WORD ;
    TL_DC_PIN_UP_LP : WORD ;
    TL_DC_PIN_DOWN_LP : WORD ;
    TL_DC_LATCH1_ADV_LP : WORD ;
    TL_DC_LATCH1_RET_LP : WORD ;
    TL_DC_LATCH2_ADV_LP : WORD ;
    TL_DC_LATCH2_RET_LP : WORD ;
    TL_DC_1ST_CLAMP1_ADV_LP : WORD ;
    TL_DC_1ST_CLAMP1_RET_LP : WORD ;
    TL_DC_1ST_CLAMP2_ADV_LP : WORD ;
    TL_DC_1ST_CLAMP2_RET_LP : WORD ;
    TL_DC_1ST_CLAMP3_ADV_LP : WORD ;
    TL_DC_1ST_CLAMP3_RET_LP : WORD ;
    TL_DC_2ND_CLAMP1_ADV_LP : WORD ;
    TL_DC_2ND_CLAMP1_RET_LP : WORD ;
    TL_DC_2ND_CLAMP2_ADV_LP : WORD ;
    TL_DC_2ND_CLAMP2_RET_LP : WORD ;
    TL_DC_U261_ADV_LP : WORD ;
    TL_DC_U261_RET_LP : WORD ;
    TL_DC_U261_CLAMP_ADV_LP : WORD ;
    TL_DC_U261_CLAMP_RET_LP : WORD ;
    TL_DC_U269_UP_LP : WORD ;
    TL_DC_U269_DOWN_LP : WORD ;
    TL_DC_U269_CLAMP_ADV_LP : WORD ;
    TL_DC_U269_CLAMP_RET_LP : WORD ;
    TL_DC_3RD_CLAMP_ADV_LP : WORD ;
    TL_DC_3RD_CLAMP_RET_LP : WORD ;
    TL_DC_U262_1_UP_LP : WORD ;
    TL_DC_U262_1_DOWN_LP : WORD ;
    TL_DC_U262_1_ADV_LP : WORD ;
    TL_DC_U262_1_RET_LP : WORD ;
    TL_DC_U262_1_CLP_ADV_LP : WORD ;
    TL_DC_U262_1_CLP_RET_LP : WORD ;
    TL_DC_U261_2_CLP_ADV_LP : WORD ;
    TL_DC_U261_2_CLP_RET_LP : WORD ;
    SP_WORD106 : WORD ;
    SP_WORD107 : WORD ;
    SP_WORD108 : WORD ;
    SP_WORD109 : WORD ;
    SP_WORD110 : WORD ;
    SP_WORD111 : WORD ;
   END_STRUCT ;
   S_704 : STRUCT
    M_AUTO_SEL : BOOL ;
    M_MANUAL_SEL : BOOL ;
    M_READY_PB : BOOL ;
    M_AUTO_RUN_PB : BOOL ;
    M_WORK_COMP_SET_PB : BOOL ;
    M_WORK_COMP_RST_PB : BOOL ;
    M_HOME_POS_PB : BOOL ;
    M_708_L_R_BT_ERR_RST : BOOL ;
    HOOK_PIN_SEL : BOOL ;
    DAECHA_LOCK_SEL : BOOL ;
    ELE_SEL : BOOL ;
    FF_CLAMP_SEL : BOOL ;
    SPARE13 : BOOL ;
    SPARE14 : BOOL ;
    SPARE15 : BOOL ;
    SPARE16 : BOOL ;
    SPARE17 : BOOL ;
    SPARE18 : BOOL ;
    SPARE19 : BOOL ;
    SPARE20 : BOOL ;
    SPARE21 : BOOL ;
    SPARE22 : BOOL ;
    SPARE23 : BOOL ;
    SPARE24 : BOOL ;
    SPARE25 : BOOL ;
    SPARE26 : BOOL ;
    SPARE27 : BOOL ;
    SPARE28 : BOOL ;
    SPARE29 : BOOL ;
    SPARE30 : BOOL ;
    M_ADV_PB : BOOL ;
    M_RET_PB : BOOL ;
    LM_DC_PIN_SEL : BOOL ;
    LM_DC_1ST_CLAMP1_SEL : BOOL ;
    LM_DC_1ST_CLAMP2_SEL : BOOL ;
    LM_DC_1ST_CLAMP3_SEL : BOOL ;
    LM_DC_1ST_CLAMP4_SEL : BOOL ;
    LM_DC_2ND_CLAMP1_SEL : BOOL ;
    LM_DC_2ND_CLAMP2_SEL : BOOL ;
    LM_DC_2ND_CLAMP3_SEL : BOOL ;
    LM_DC_2ND_CLAMP4_SEL : BOOL ;
    LM_DC_2ND_CLAMP5_SEL : BOOL ;
    LM_DC_DR_STK_PIN_SEL : BOOL ;
    LM_DC_OTR_CLAMP_SEL : BOOL ;
    LM_DC_ASSY_CLAMP_SEL : BOOL ;
    LM_DC_FF_PIN_SEL : BOOL ;
    LM_DC_FF_CLAMP_SEL : BOOL ;
    LM_DC_2ND_CLAMP6_SEL : BOOL ;
    SPARE50 : BOOL ;
    SPARE51 : BOOL ;
    SPARE52 : BOOL ;
    SPARE53 : BOOL ;
    SPARE54 : BOOL ;
    SPARE55 : BOOL ;
    SPARE56 : BOOL ;
    SPARE57 : BOOL ;
    SPARE58 : BOOL ;
    SPARE59 : BOOL ;
    SPARE60 : BOOL ;
    SPARE61 : BOOL ;
    SPARE62 : BOOL ;
    SPARE63 : BOOL ;
    LM_DC_M_ADV_PB : BOOL ;
    LM_DC_M_RET_PB : BOOL ;
    TL_DC_PIN_SEL : BOOL ;
    TL_DC_LATCH1_SEL : BOOL ;
    TL_DC_1ST_CLAMP_SEL : BOOL ;
    TL_DC_2ND_CLAMP_SEL : BOOL ;
    TL_DC_U261_SEL : BOOL ;
    TL_DC_U261_CLAMP_SEL : BOOL ;
    TL_DC_U269_UP_DN_SEL : BOOL ;
    TL_DC_U269_CLAMP_SEL : BOOL ;
    TL_DC_3RD_CLAMP_SEL : BOOL ;
    TL_DC_U262_1_UP_DN_SEL : BOOL ;
    TL_DC_U262_1_SEL : BOOL ;
    TL_DC_U262_1_CLAMP_SEL : BOOL ;
    TL_DC_U261_2_CLAMP_SEL : BOOL ;
    SPARE79 : BOOL ;
    SPARE80 : BOOL ;
    SPARE81 : BOOL ;
    SPARE82 : BOOL ;
    SPARE83 : BOOL ;
    SPARE84 : BOOL ;
    SPARE85 : BOOL ;
    SPARE86 : BOOL ;
    SPARE87 : BOOL ;
    SPARE88 : BOOL ;
    SPARE89 : BOOL ;
    SPARE90 : BOOL ;
    SPARE91 : BOOL ;
    SPARE92 : BOOL ;
    SPARE93 : BOOL ;
    SPARE94 : BOOL ;
    SPARE95 : BOOL ;
    TL_DC_M_ADV_PB : BOOL ;
    TL_DC_M_RET_PB : BOOL ;
    SPARE98 : BOOL ;
    SPARE99 : BOOL ;
    SPARE100 : BOOL ;
    SPARE101 : BOOL ;
    SPARE102 : BOOL ;
    SPARE103 : BOOL ;
    SPARE104 : BOOL ;
    SPARE105 : BOOL ;
    SPARE106 : BOOL ;
    SPARE107 : BOOL ;
    SPARE108 : BOOL ;
    SPARE109 : BOOL ;
    SPARE110 : BOOL ;
    SPARE111 : BOOL ;
    SPARE112 : BOOL ;
    SPARE113 : BOOL ;
    SPARE114 : BOOL ;
    SPARE115 : BOOL ;
    SPARE116 : BOOL ;
    SPARE117 : BOOL ;
    SPARE118 : BOOL ;
    SPARE119 : BOOL ;
    SPARE120 : BOOL ;
    SPARE121 : BOOL ;
    SPARE122 : BOOL ;
    SPARE123 : BOOL ;
    SPARE124 : BOOL ;
    SPARE125 : BOOL ;
    SPARE126 : BOOL ;
    SPARE127 : BOOL ;
    SPARE128 : BOOL ;
    SPARE129 : BOOL ;
    SP_WORD1 : WORD ;
    SP_WORD2 : WORD ;
    HOOK_PIN_UP_LP : WORD ;
    HOOK_PIN_DOWN_LP : WORD ;
    DAECHA_LOCK_ADV_LP : WORD ;
    DAECHA_LOCK_RET_LP : WORD ;
    ELE_ADV_LP : WORD ;
    ELE_RET_LP : WORD ;
    AIR_ELE_ADV_LP : WORD ;
    AIR_ELE_RET_LP : WORD ;
    FF_CLAMP_ADV_LP : WORD ;
    FF_CLAMP_RET_LP : WORD ;
    LM_DC_PIN_UP_LP : WORD ;
    LM_DC_PIN_DOWN_LP : WORD ;
    LM_DC_1ST_CLAMP1_ADV_LP : WORD ;
    LM_DC_1ST_CLAMP1_RET_LP : WORD ;
    LM_DC_1ST_CLAMP2_ADV_LP : WORD ;
    LM_DC_1ST_CLAMP2_RET_LP : WORD ;
    LM_DC_1ST_CLAMP3_ADV_LP : WORD ;
    LM_DC_1ST_CLAMP3_RET_LP : WORD ;
    LM_DC_1ST_CLAMP4_ADV_LP : WORD ;
    LM_DC_1ST_CLAMP4_RET_LP : WORD ;
    LM_DC_2ND_CLAMP1_ADV_LP : WORD ;
    LM_DC_2ND_CLAMP1_RET_LP : WORD ;
    LM_DC_2ND_CLAMP2_ADV_LP : WORD ;
    LM_DC_2ND_CLAMP2_RET_LP : WORD ;
    LM_DC_2ND_CLAMP3_ADV_LP : WORD ;
    LM_DC_2ND_CLAMP3_RET_LP : WORD ;
    LM_DC_2ND_CLAMP4_ADV_LP : WORD ;
    LM_DC_2ND_CLAMP4_RET_LP : WORD ;
    LM_DC_2ND_CLAMP5_ADV_LP : WORD ;
    LM_DC_2ND_CLAMP5_RET_LP : WORD ;
    LM_DC_DR_STK_PIN_UP_LP : WORD ;
    LM_DC_DR_STK_PIN_DOWN_LP : WORD ;
    LM_DC_OTR_CLAMP_ADV_LP : WORD ;
    LM_DC_OTR_CLAMP_RET_LP : WORD ;
    LM_DC_ASSY_CLAMP_ADV_LP : WORD ;
    LM_DC_ASSY_CLAMP_RET_LP : WORD ;
    LM_DC_FF_PIN_UP_LP : WORD ;
    LM_DC_FF_PIN_DOWN_LP : WORD ;
    LM_DC_FF_CLAMP_ADV_LP : WORD ;
    LM_DC_FF_CLAMP_RET_LP : WORD ;
    LM_DC_2ND_CLAMP6_ADV_LP : WORD ;
    LM_DC_2ND_CLAMP6_RET_LP : WORD ;
    LM_DC_2ND_CLAMP7_ADV_LP : WORD ;
    LM_DC_2ND_CLAMP7_RET_LP : WORD ;
    LM_DC_1ST_CLAMP5_ADV_LP : WORD ;
    LM_DC_1ST_CLAMP5_RET_LP : WORD ;
    SP_WORD68 : WORD ;
    SP_WORD69 : WORD ;
    SP_WORD70 : WORD ;
    SP_WORD71 : WORD ;
    TL_DC_PIN_UP_LP : WORD ;
    TL_DC_PIN_DOWN_LP : WORD ;
    TL_DC_LATCH1_ADV_LP : WORD ;
    TL_DC_LATCH1_RET_LP : WORD ;
    TL_DC_LATCH2_ADV_LP : WORD ;
    TL_DC_LATCH2_RET_LP : WORD ;
    TL_DC_1ST_CLAMP1_ADV_LP : WORD ;
    TL_DC_1ST_CLAMP1_RET_LP : WORD ;
    TL_DC_1ST_CLAMP2_ADV_LP : WORD ;
    TL_DC_1ST_CLAMP2_RET_LP : WORD ;
    TL_DC_1ST_CLAMP3_ADV_LP : WORD ;
    TL_DC_1ST_CLAMP3_RET_LP : WORD ;
    TL_DC_2ND_CLAMP1_ADV_LP : WORD ;
    TL_DC_2ND_CLAMP1_RET_LP : WORD ;
    TL_DC_2ND_CLAMP2_ADV_LP : WORD ;
    TL_DC_2ND_CLAMP2_RET_LP : WORD ;
    TL_DC_U261_ADV_LP : WORD ;
    TL_DC_U261_RET_LP : WORD ;
    TL_DC_U261_CLAMP_ADV_LP : WORD ;
    TL_DC_U261_CLAMP_RET_LP : WORD ;
    TL_DC_U269_UP_LP : WORD ;
    TL_DC_U269_DOWN_LP : WORD ;
    TL_DC_U269_CLAMP_ADV_LP : WORD ;
    TL_DC_U269_CLAMP_RET_LP : WORD ;
    TL_DC_3RD_CLAMP_ADV_LP : WORD ;
    TL_DC_3RD_CLAMP_RET_LP : WORD ;
    TL_DC_U262_1_UP_LP : WORD ;
    TL_DC_U262_1_DOWN_LP : WORD ;
    TL_DC_U262_1_ADV_LP : WORD ;
    TL_DC_U262_1_RET_LP : WORD ;
    TL_DC_U262_1_CLP_ADV_LP : WORD ;
    TL_DC_U262_1_CLP_RET_LP : WORD ;
    TL_DC_U261_2_CLP_ADV_LP : WORD ;
    TL_DC_U261_2_CLP_RET_LP : WORD ;
    SP_WORD106 : WORD ;
    SP_WORD107 : WORD ;
    SP_WORD108 : WORD ;
    SP_WORD109 : WORD ;
    AIR_ELE_AR_ADV_LP : WORD ;
    AIR_ELE_AR_RET_LP : WORD ;
   END_STRUCT ;
   S_DOWNDL : STRUCT
    M_AUTO_SEL : BOOL ;
    M_MANUAL_SEL : BOOL ;
    M_READY_PB : BOOL ;
    M_AUTO_RUN_PB : BOOL ;
    M_WORK_COMP_SET_PB : BOOL ;
    M_WORK_COMP_RST_PB : BOOL ;
    M_HOME_POS_PB : BOOL ;
    SPARE8 : BOOL ;
    DAECHA_IN_SEL : BOOL ;
    DAECHA_OUT_SEL : BOOL ;
    DAECHA_CLAMP_SEL : BOOL ;
    LIFT_LOCK_SEL : BOOL ;
    LIFT_SEL : BOOL ;
    SPARE14 : BOOL ;
    SPARE15 : BOOL ;
    SPARE16 : BOOL ;
    SPARE17 : BOOL ;
    SPARE18 : BOOL ;
    SPARE19 : BOOL ;
    SPARE20 : BOOL ;
    SPARE21 : BOOL ;
    SPARE22 : BOOL ;
    SPARE23 : BOOL ;
    SPARE24 : BOOL ;
    SPARE25 : BOOL ;
    SPARE26 : BOOL ;
    SPARE27 : BOOL ;
    SPARE28 : BOOL ;
    SPARE29 : BOOL ;
    SPARE30 : BOOL ;
    M_ADV_PB : BOOL ;
    M_RET_PB : BOOL ;
    SPARE34 : BOOL ;
    SPARE35 : BOOL ;
    SPARE36 : BOOL ;
    SPARE37 : BOOL ;
    SPARE38 : BOOL ;
    SPARE39 : BOOL ;
    SPARE40 : BOOL ;
    SPARE41 : BOOL ;
    SPARE42 : BOOL ;
    SPARE43 : BOOL ;
    SPARE44 : BOOL ;
    SPARE45 : BOOL ;
    SPARE46 : BOOL ;
    SPARE47 : BOOL ;
    SPARE48 : BOOL ;
    SPARE49 : BOOL ;
    SPARE50 : BOOL ;
    SPARE51 : BOOL ;
    SPARE52 : BOOL ;
    SPARE53 : BOOL ;
    SPARE54 : BOOL ;
    SPARE55 : BOOL ;
    SPARE56 : BOOL ;
    SPARE57 : BOOL ;
    SPARE58 : BOOL ;
    SPARE59 : BOOL ;
    SPARE60 : BOOL ;
    SPARE61 : BOOL ;
    SPARE62 : BOOL ;
    SPARE63 : BOOL ;
    SPARE64 : BOOL ;
    SPARE65 : BOOL ;
    SPARE66 : BOOL ;
    SPARE67 : BOOL ;
    SPARE68 : BOOL ;
    SPARE69 : BOOL ;
    SPARE70 : BOOL ;
    SPARE71 : BOOL ;
    SPARE72 : BOOL ;
    SPARE73 : BOOL ;
    SPARE74 : BOOL ;
    SPARE75 : BOOL ;
    SPARE76 : BOOL ;
    SPARE77 : BOOL ;
    SPARE78 : BOOL ;
    SPARE79 : BOOL ;
    SPARE80 : BOOL ;
    SPARE81 : BOOL ;
    SPARE82 : BOOL ;
    SPARE83 : BOOL ;
    SPARE84 : BOOL ;
    SPARE85 : BOOL ;
    SPARE86 : BOOL ;
    SPARE87 : BOOL ;
    SPARE88 : BOOL ;
    SPARE89 : BOOL ;
    SPARE90 : BOOL ;
    SPARE91 : BOOL ;
    SPARE92 : BOOL ;
    SPARE93 : BOOL ;
    SPARE94 : BOOL ;
    SPARE95 : BOOL ;
    SPARE96 : BOOL ;
    SPARE97 : BOOL ;
    SPARE98 : BOOL ;
    SPARE99 : BOOL ;
    SPARE100 : BOOL ;
    SPARE101 : BOOL ;
    SPARE102 : BOOL ;
    SPARE103 : BOOL ;
    SPARE104 : BOOL ;
    SPARE105 : BOOL ;
    SPARE106 : BOOL ;
    SPARE107 : BOOL ;
    SPARE108 : BOOL ;
    SPARE109 : BOOL ;
    SPARE110 : BOOL ;
    SPARE111 : BOOL ;
    SPARE112 : BOOL ;
    SPARE113 : BOOL ;
    SPARE114 : BOOL ;
    SPARE115 : BOOL ;
    SPARE116 : BOOL ;
    SPARE117 : BOOL ;
    SPARE118 : BOOL ;
    SPARE119 : BOOL ;
    SPARE120 : BOOL ;
    SPARE121 : BOOL ;
    SPARE122 : BOOL ;
    SPARE123 : BOOL ;
    SPARE124 : BOOL ;
    SPARE125 : BOOL ;
    SPARE126 : BOOL ;
    SPARE127 : BOOL ;
    SPARE128 : BOOL ;
    SPARE129 : BOOL ;
    SPARE130 : BOOL ;
    SPARE131 : BOOL ;
    SPARE132 : BOOL ;
    SPARE133 : BOOL ;
    SPARE134 : BOOL ;
    SPARE135 : BOOL ;
    SPARE136 : BOOL ;
    SPARE137 : BOOL ;
    SPARE138 : BOOL ;
    SPARE139 : BOOL ;
    SPARE140 : BOOL ;
    SPARE141 : BOOL ;
    SPARE142 : BOOL ;
    SPARE143 : BOOL ;
    SPARE144 : BOOL ;
    SPARE145 : BOOL ;
    SPARE146 : BOOL ;
    SPARE147 : BOOL ;
    SPARE148 : BOOL ;
    SPARE149 : BOOL ;
    SPARE150 : BOOL ;
    SPARE151 : BOOL ;
    SPARE152 : BOOL ;
    SPARE153 : BOOL ;
    SPARE154 : BOOL ;
    SPARE155 : BOOL ;
    SPARE156 : BOOL ;
    SPARE157 : BOOL ;
    SPARE158 : BOOL ;
    SPARE159 : BOOL ;
    SPARE160 : BOOL ;
    SPARE161 : BOOL ;
    DAECHA_IN_ADV_LP : WORD ;
    DAECHA_IN_RET_LP : WORD ;
    DAECHA_OUT_ADV_LP : WORD ;
    DAECHA_OUT_RET_LP : WORD ;
    DAECHA_CLAMP_ADV_LP : WORD ;
    DAECHA_CLAMP_RET_LP : WORD ;
    LIFT_LOCK_ADV_LP : WORD ;
    LIFT_LOCK_RET_LP : WORD ;
    LIFT_UP_LP : WORD ;
    LIFT_DOWN_LP : WORD ;
    SP_WORD21 : WORD ;
    SP_WORD22 : WORD ;
    SP_WORD23 : WORD ;
    SP_WORD24 : WORD ;
    SP_WORD25 : WORD ;
    SP_WORD26 : WORD ;
    SP_WORD27 : WORD ;
    SP_WORD28 : WORD ;
    SP_WORD29 : WORD ;
    SP_WORD30 : WORD ;
    SP_WORD31 : WORD ;
    SP_WORD32 : WORD ;
    SP_WORD33 : WORD ;
    SP_WORD34 : WORD ;
    SP_WORD35 : WORD ;
    SP_WORD36 : WORD ;
    SP_WORD37 : WORD ;
    SP_WORD38 : WORD ;
    SP_WORD39 : WORD ;
    SP_WORD40 : WORD ;
    SP_WORD41 : WORD ;
    SP_WORD42 : WORD ;
    SP_WORD43 : WORD ;
    SP_WORD44 : WORD ;
    SP_WORD45 : WORD ;
    SP_WORD46 : WORD ;
    SP_WORD47 : WORD ;
    SP_WORD49 : WORD ;
    SP_WORD50 : WORD ;
    SP_WORD51 : WORD ;
    SP_WORD52 : WORD ;
    SP_WORD53 : WORD ;
    SP_WORD54 : WORD ;
    SP_WORD55 : WORD ;
    SP_WORD56 : WORD ;
    SP_WORD57 : WORD ;
    SP_WORD58 : WORD ;
    SP_WORD59 : WORD ;
    SP_WORD60 : WORD ;
    SP_WORD61 : WORD ;
    SP_WORD62 : WORD ;
    SP_WORD63 : WORD ;
    SP_WORD64 : WORD ;
    SP_WORD65 : WORD ;
    SP_WORD66 : WORD ;
    SP_WORD67 : WORD ;
    SP_WORD68 : WORD ;
    SP_WORD69 : WORD ;
    SP_WORD70 : WORD ;
    SP_WORD71 : WORD ;
    SP_WORD72 : WORD ;
    SP_WORD73 : WORD ;
    SP_WORD74 : WORD ;
    SP_WORD75 : WORD ;
    SP_WORD76 : WORD ;
    SP_WORD77 : WORD ;
    SP_WORD78 : WORD ;
    SP_WORD79 : WORD ;
    SP_WORD80 : WORD ;
    SP_WORD81 : WORD ;
    SP_WORD82 : WORD ;
    SP_WORD83 : WORD ;
    SP_WORD84 : WORD ;
    SP_WORD85 : WORD ;
    SP_WORD86 : WORD ;
    SP_WORD87 : WORD ;
    SP_WORD88 : WORD ;
    SP_WORD89 : WORD ;
    SP_WORD90 : WORD ;
    SP_WORD91 : WORD ;
    SP_WORD92 : WORD ;
    SP_WORD93 : WORD ;
    SP_WORD94 : WORD ;
    SP_WORD95 : WORD ;
    SP_WORD96 : WORD ;
    SP_WORD97 : WORD ;
    SP_WORD98 : WORD ;
    SP_WORD99 : WORD ;
    SP_WORD100 : WORD ;
    SP_WORD101 : WORD ;
   END_STRUCT ;
   S_ROOF_RACK : STRUCT
    M_AUTO_SEL : BOOL ;
    M_MANUAL_SEL : BOOL ;
    M_READY_PB : BOOL ;
    M_AUTO_RUN_PB : BOOL ;
    M_WORK_COMP_SET_PB : BOOL ;
    M_WORK_COMP_RST_PB : BOOL ;
    M_HOME_POS_PB : BOOL ;
    SPARE8 : BOOL ;
    ROOF_RACK_ADV_RET_SEL : BOOL ;
    ROOF_RACK_CLAMP_SEL : BOOL ;
    ROOF_RACK_GUN1_A_R_SEL : BOOL ;
    ROOF_RACK_GUN2_A_R_SEL : BOOL ;
    ROOF_RACK_GUN1_PRESS_SEL : BOOL ;
    ROOF_RACK_GUN2_PRESS_SEL : BOOL ;
    ROOF_RACK_WELD_ON_SEL : BOOL ;
    SPARE16 : BOOL ;
    SPARE17 : BOOL ;
    SPARE18 : BOOL ;
    SPARE19 : BOOL ;
    SPARE20 : BOOL ;
    SPARE21 : BOOL ;
    SPARE22 : BOOL ;
    SPARE23 : BOOL ;
    SPARE24 : BOOL ;
    SPARE25 : BOOL ;
    SPARE26 : BOOL ;
    SPARE27 : BOOL ;
    SPARE28 : BOOL ;
    SPARE29 : BOOL ;
    SPARE30 : BOOL ;
    M_ADV_PB : BOOL ;
    M_RET_PB : BOOL ;
    SPARE34 : BOOL ;
    SPARE35 : BOOL ;
    SPARE36 : BOOL ;
    SPARE37 : BOOL ;
    SPARE38 : BOOL ;
    SPARE39 : BOOL ;
    SPARE40 : BOOL ;
    SPARE41 : BOOL ;
    SPARE42 : BOOL ;
    SPARE43 : BOOL ;
    SPARE44 : BOOL ;
    SPARE45 : BOOL ;
    SPARE46 : BOOL ;
    SPARE47 : BOOL ;
    SPARE48 : BOOL ;
    SPARE49 : BOOL ;
    SPARE50 : BOOL ;
    SPARE51 : BOOL ;
    SPARE52 : BOOL ;
    SPARE53 : BOOL ;
    SPARE54 : BOOL ;
    SPARE55 : BOOL ;
    SPARE56 : BOOL ;
    SPARE57 : BOOL ;
    SPARE58 : BOOL ;
    SPARE59 : BOOL ;
    SPARE60 : BOOL ;
    SPARE61 : BOOL ;
    SPARE62 : BOOL ;
    SPARE63 : BOOL ;
    SPARE64 : BOOL ;
    SPARE65 : BOOL ;
    SPARE66 : BOOL ;
    SPARE67 : BOOL ;
    SPARE68 : BOOL ;
    SPARE69 : BOOL ;
    SPARE70 : BOOL ;
    SPARE71 : BOOL ;
    SPARE72 : BOOL ;
    SPARE73 : BOOL ;
    SPARE74 : BOOL ;
    SPARE75 : BOOL ;
    SPARE76 : BOOL ;
    SPARE77 : BOOL ;
    SPARE78 : BOOL ;
    SPARE79 : BOOL ;
    SPARE80 : BOOL ;
    SPARE81 : BOOL ;
    SPARE82 : BOOL ;
    SPARE83 : BOOL ;
    SPARE84 : BOOL ;
    SPARE85 : BOOL ;
    SPARE86 : BOOL ;
    SPARE87 : BOOL ;
    SPARE88 : BOOL ;
    SPARE89 : BOOL ;
    SPARE90 : BOOL ;
    SPARE91 : BOOL ;
    SPARE92 : BOOL ;
    SPARE93 : BOOL ;
    SPARE94 : BOOL ;
    SPARE95 : BOOL ;
    SPARE96 : BOOL ;
    SPARE97 : BOOL ;
    SPARE98 : BOOL ;
    SPARE99 : BOOL ;
    SPARE100 : BOOL ;
    SPARE101 : BOOL ;
    SPARE102 : BOOL ;
    SPARE103 : BOOL ;
    SPARE104 : BOOL ;
    SPARE105 : BOOL ;
    SPARE106 : BOOL ;
    SPARE107 : BOOL ;
    SPARE108 : BOOL ;
    SPARE109 : BOOL ;
    SPARE110 : BOOL ;
    SPARE111 : BOOL ;
    SPARE112 : BOOL ;
    SPARE113 : BOOL ;
    SPARE114 : BOOL ;
    SPARE115 : BOOL ;
    SPARE116 : BOOL ;
    SPARE117 : BOOL ;
    SPARE118 : BOOL ;
    SPARE119 : BOOL ;
    SPARE120 : BOOL ;
    SPARE121 : BOOL ;
    SPARE122 : BOOL ;
    SPARE123 : BOOL ;
    SPARE124 : BOOL ;
    SPARE125 : BOOL ;
    SPARE126 : BOOL ;
    SPARE127 : BOOL ;
    SPARE128 : BOOL ;
    SPARE129 : BOOL ;
    SPARE130 : BOOL ;
    SPARE131 : BOOL ;
    SPARE132 : BOOL ;
    SPARE133 : BOOL ;
    SPARE134 : BOOL ;
    SPARE135 : BOOL ;
    SPARE136 : BOOL ;
    SPARE137 : BOOL ;
    SPARE138 : BOOL ;
    SPARE139 : BOOL ;
    SPARE140 : BOOL ;
    SPARE141 : BOOL ;
    SPARE142 : BOOL ;
    SPARE143 : BOOL ;
    SPARE144 : BOOL ;
    SPARE145 : BOOL ;
    SPARE146 : BOOL ;
    SPARE147 : BOOL ;
    SPARE148 : BOOL ;
    SPARE149 : BOOL ;
    SPARE150 : BOOL ;
    SPARE151 : BOOL ;
    SPARE152 : BOOL ;
    SPARE153 : BOOL ;
    SPARE154 : BOOL ;
    SPARE155 : BOOL ;
    SPARE156 : BOOL ;
    SPARE157 : BOOL ;
    SPARE158 : BOOL ;
    SPARE159 : BOOL ;
    SPARE160 : BOOL ;
    SPARE161 : BOOL ;
    ROOF_RACK_ADV_LP : WORD ;
    ROOF_RACK_RET_LP : WORD ;
    ROOF_RACK_CLAMP_ADV_LP : WORD ;
    ROOF_RACK_CLAMP_RET_LP : WORD ;
    ROOF_RACK_GUN1_ADV_LP : WORD ;
    ROOF_RACK_GUN1_RET_LP : WORD ;
    ROOF_RACK_GUN2_ADV_LP : WORD ;
    ROOF_RACK_GUN2_RET_LP : WORD ;
    ROOF_RACK_GUN1_PRESS_LP : WORD ;
    ROOF_RACK_GUN1_OPEN_LP : WORD ;
    ROOF_RACK_GUN2_PRESS_LP : WORD ;
    ROOF_RACK_GUN2_OPEN_LP : WORD ;
    SP_WORD23 : WORD ;
    SP_WORD24 : WORD ;
    SP_WORD25 : WORD ;
    SP_WORD26 : WORD ;
    SP_WORD27 : WORD ;
    SP_WORD28 : WORD ;
    SP_WORD29 : WORD ;
    SP_WORD30 : WORD ;
    SP_WORD31 : WORD ;
    SP_WORD32 : WORD ;
    SP_WORD33 : WORD ;
    SP_WORD34 : WORD ;
    SP_WORD35 : WORD ;
    SP_WORD36 : WORD ;
    SP_WORD37 : WORD ;
    SP_WORD38 : WORD ;
    SP_WORD39 : WORD ;
    SP_WORD40 : WORD ;
    SP_WORD41 : WORD ;
    SP_WORD42 : WORD ;
    SP_WORD43 : WORD ;
    SP_WORD44 : WORD ;
    SP_WORD45 : WORD ;
    SP_WORD46 : WORD ;
    SP_WORD47 : WORD ;
    SP_WORD49 : WORD ;
    SP_WORD50 : WORD ;
    SP_WORD51 : WORD ;
    SP_WORD52 : WORD ;
    SP_WORD53 : WORD ;
    SP_WORD54 : WORD ;
    SP_WORD55 : WORD ;
    SP_WORD56 : WORD ;
    SP_WORD57 : WORD ;
    SP_WORD58 : WORD ;
    SP_WORD59 : WORD ;
    SP_WORD60 : WORD ;
    SP_WORD61 : WORD ;
    SP_WORD62 : WORD ;
    SP_WORD63 : WORD ;
    SP_WORD64 : WORD ;
    SP_WORD65 : WORD ;
    SP_WORD66 : WORD ;
    SP_WORD67 : WORD ;
    SP_WORD68 : WORD ;
    SP_WORD69 : WORD ;
    SP_WORD70 : WORD ;
    SP_WORD71 : WORD ;
    SP_WORD72 : WORD ;
    SP_WORD73 : WORD ;
    SP_WORD74 : WORD ;
    SP_WORD75 : WORD ;
    SP_WORD76 : WORD ;
    SP_WORD77 : WORD ;
    SP_WORD78 : WORD ;
    SP_WORD79 : WORD ;
    SP_WORD80 : WORD ;
    SP_WORD81 : WORD ;
    SP_WORD82 : WORD ;
    SP_WORD83 : WORD ;
    SP_WORD84 : WORD ;
    SP_WORD85 : WORD ;
    SP_WORD86 : WORD ;
    SP_WORD87 : WORD ;
    SP_WORD88 : WORD ;
    SP_WORD89 : WORD ;
    SP_WORD90 : WORD ;
    SP_WORD91 : WORD ;
    SP_WORD92 : WORD ;
    SP_WORD93 : WORD ;
    SP_WORD94 : WORD ;
    SP_WORD95 : WORD ;
    SP_WORD96 : WORD ;
    SP_WORD97 : WORD ;
    SP_WORD98 : WORD ;
    SP_WORD99 : WORD ;
    SP_WORD100 : WORD ;
    SP_WORD101 : WORD ;
   END_STRUCT ;
  END_STRUCT ;
BEGIN
   S_SHUTTLE.M_AUTO_SEL := FALSE;
   S_SHUTTLE.M_MANUAL_SEL := FALSE;
   S_SHUTTLE.M_READY_PB := FALSE;
   S_SHUTTLE.M_AUTO_RUN_PB := FALSE;
   S_SHUTTLE.M_WORK_COMP_SET_PB := FALSE;
   S_SHUTTLE.M_WORK_COMP_RST_PB := FALSE;
   S_SHUTTLE.M_HOME_POS_PB := FALSE;
   S_SHUTTLE.M_TIP_DRESS_PB := FALSE;
   S_SHUTTLE.HOOK_PIN_SEL := FALSE;
   S_SHUTTLE.DAECHA_LOCK_SEL := FALSE;
   S_SHUTTLE.ELE_SEL := FALSE;
   S_SHUTTLE.AIR_ELE_SEL := FALSE;
   S_SHUTTLE.SPARE13 := FALSE;
   S_SHUTTLE.SPARE14 := FALSE;
   S_SHUTTLE.SPARE15 := FALSE;
   S_SHUTTLE.M_ALL_TIP_DRESS_PB := FALSE;
   S_SHUTTLE.SPARE17 := FALSE;
   S_SHUTTLE.SPARE18 := FALSE;
   S_SHUTTLE.SPARE19 := FALSE;
   S_SHUTTLE.SPARE20 := FALSE;
   S_SHUTTLE.SPARE21 := FALSE;
   S_SHUTTLE.SPARE22 := FALSE;
   S_SHUTTLE.SPARE23 := FALSE;
   S_SHUTTLE.SPARE24 := FALSE;
   S_SHUTTLE.SERVO_LOW_SS := FALSE;
   S_SHUTTLE.SERVO_HIGH_SS := FALSE;
   S_SHUTTLE.MELODY_ON_PB := FALSE;
   S_SHUTTLE.SPARE28 := FALSE;
   S_SHUTTLE.SPARE29 := FALSE;
   S_SHUTTLE.SPARE30 := FALSE;
   S_SHUTTLE.M_ADV_PB := FALSE;
   S_SHUTTLE.M_RET_PB := FALSE;
   S_SHUTTLE.SPARE33 := FALSE;
   S_SHUTTLE.SPARE34 := FALSE;
   S_SHUTTLE.SPARE35 := FALSE;
   S_SHUTTLE.SPARE36 := FALSE;
   S_SHUTTLE.SPARE37 := FALSE;
   S_SHUTTLE.SPARE38 := FALSE;
   S_SHUTTLE.SPARE39 := FALSE;
   S_SHUTTLE.SPARE40 := FALSE;
   S_SHUTTLE.SPARE41 := FALSE;
   S_SHUTTLE.SPARE42 := FALSE;
   S_SHUTTLE.SPARE43 := FALSE;
   S_SHUTTLE.SPARE44 := FALSE;
   S_SHUTTLE.SPARE45 := FALSE;
   S_SHUTTLE.SPARE46 := FALSE;
   S_SHUTTLE.SPARE47 := FALSE;
   S_SHUTTLE.SPARE48 := FALSE;
   S_SHUTTLE.SPARE50 := FALSE;
   S_SHUTTLE.SPARE51 := FALSE;
   S_SHUTTLE.SPARE52 := FALSE;
   S_SHUTTLE.SPARE53 := FALSE;
   S_SHUTTLE.SPARE54 := FALSE;
   S_SHUTTLE.SPARE55 := FALSE;
   S_SHUTTLE.SPARE56 := FALSE;
   S_SHUTTLE.SPARE57 := FALSE;
   S_SHUTTLE.SPARE58 := FALSE;
   S_SHUTTLE.SPARE59 := FALSE;
   S_SHUTTLE.SPARE60 := FALSE;
   S_SHUTTLE.SPARE61 := FALSE;
   S_SHUTTLE.SPARE62 := FALSE;
   S_SHUTTLE.SPARE63 := FALSE;
   S_SHUTTLE.SPARE64 := FALSE;
   S_SHUTTLE.SPARE65 := FALSE;
   S_SHUTTLE.SPARE66 := FALSE;
   S_SHUTTLE.SPARE67 := FALSE;
   S_SHUTTLE.SPARE68 := FALSE;
   S_SHUTTLE.SPARE69 := FALSE;
   S_SHUTTLE.SPARE70 := FALSE;
   S_SHUTTLE.SPARE71 := FALSE;
   S_SHUTTLE.SPARE72 := FALSE;
   S_SHUTTLE.SPARE73 := FALSE;
   S_SHUTTLE.SPARE74 := FALSE;
   S_SHUTTLE.SPARE75 := FALSE;
   S_SHUTTLE.SPARE76 := FALSE;
   S_SHUTTLE.SPARE77 := FALSE;
   S_SHUTTLE.SPARE78 := FALSE;
   S_SHUTTLE.SPARE79 := FALSE;
   S_SHUTTLE.SPARE80 := FALSE;
   S_SHUTTLE.SPARE81 := FALSE;
   S_SHUTTLE.SPARE82 := FALSE;
   S_SHUTTLE.SPARE83 := FALSE;
   S_SHUTTLE.SPARE84 := FALSE;
   S_SHUTTLE.SPARE85 := FALSE;
   S_SHUTTLE.SPARE86 := FALSE;
   S_SHUTTLE.SPARE87 := FALSE;
   S_SHUTTLE.SPARE88 := FALSE;
   S_SHUTTLE.SPARE89 := FALSE;
   S_SHUTTLE.SPARE90 := FALSE;
   S_SHUTTLE.SPARE91 := FALSE;
   S_SHUTTLE.SPARE92 := FALSE;
   S_SHUTTLE.SPARE93 := FALSE;
   S_SHUTTLE.SPARE94 := FALSE;
   S_SHUTTLE.SPARE95 := FALSE;
   S_SHUTTLE.SPARE96 := FALSE;
   S_SHUTTLE.SPARE97 := FALSE;
   S_SHUTTLE.SPARE98 := FALSE;
   S_SHUTTLE.SPARE99 := FALSE;
   S_SHUTTLE.SPARE100 := FALSE;
   S_SHUTTLE.SPARE101 := FALSE;
   S_SHUTTLE.SPARE102 := FALSE;
   S_SHUTTLE.SPARE103 := FALSE;
   S_SHUTTLE.SPARE104 := FALSE;
   S_SHUTTLE.SPARE105 := FALSE;
   S_SHUTTLE.SPARE106 := FALSE;
   S_SHUTTLE.SPARE107 := FALSE;
   S_SHUTTLE.SPARE108 := FALSE;
   S_SHUTTLE.SPARE109 := FALSE;
   S_SHUTTLE.SPARE110 := FALSE;
   S_SHUTTLE.SPARE111 := FALSE;
   S_SHUTTLE.SPARE112 := FALSE;
   S_SHUTTLE.SPARE113 := FALSE;
   S_SHUTTLE.SPARE114 := FALSE;
   S_SHUTTLE.SPARE115 := FALSE;
   S_SHUTTLE.SPARE116 := FALSE;
   S_SHUTTLE.SPARE117 := FALSE;
   S_SHUTTLE.SPARE118 := FALSE;
   S_SHUTTLE.SPARE119 := FALSE;
   S_SHUTTLE.SPARE120 := FALSE;
   S_SHUTTLE.SPARE121 := FALSE;
   S_SHUTTLE.SPARE122 := FALSE;
   S_SHUTTLE.SPARE123 := FALSE;
   S_SHUTTLE.SPARE124 := FALSE;
   S_SHUTTLE.SPARE125 := FALSE;
   S_SHUTTLE.SPARE126 := FALSE;
   S_SHUTTLE.SPARE127 := FALSE;
   S_SHUTTLE.SPARE128 := FALSE;
   S_SHUTTLE.SPARE129 := FALSE;
   S_SHUTTLE.SPARE130 := FALSE;
   S_SHUTTLE.SPARE131 := FALSE;
   S_SHUTTLE.SPARE132 := FALSE;
   S_SHUTTLE.SPARE133 := FALSE;
   S_SHUTTLE.SPARE134 := FALSE;
   S_SHUTTLE.SPARE135 := FALSE;
   S_SHUTTLE.SPARE136 := FALSE;
   S_SHUTTLE.SPARE137 := FALSE;
   S_SHUTTLE.SPARE138 := FALSE;
   S_SHUTTLE.SPARE139 := FALSE;
   S_SHUTTLE.SPARE140 := FALSE;
   S_SHUTTLE.SPARE141 := FALSE;
   S_SHUTTLE.SPARE142 := FALSE;
   S_SHUTTLE.SPARE143 := FALSE;
   S_SHUTTLE.SPARE144 := FALSE;
   S_SHUTTLE.SPARE145 := FALSE;
   S_SHUTTLE.SPARE146 := FALSE;
   S_SHUTTLE.SPARE147 := FALSE;
   S_SHUTTLE.SPARE148 := FALSE;
   S_SHUTTLE.SPARE149 := FALSE;
   S_SHUTTLE.SPARE150 := FALSE;
   S_SHUTTLE.SPARE151 := FALSE;
   S_SHUTTLE.SPARE152 := FALSE;
   S_SHUTTLE.SPARE153 := FALSE;
   S_SHUTTLE.SPARE154 := FALSE;
   S_SHUTTLE.SPARE155 := FALSE;
   S_SHUTTLE.SPARE156 := FALSE;
   S_SHUTTLE.SPARE157 := FALSE;
   S_SHUTTLE.SPARE158 := FALSE;
   S_SHUTTLE.SPARE159 := FALSE;
   S_SHUTTLE.SPARE160 := FALSE;
   S_SHUTTLE.SPARE161 := FALSE;
   S_SHUTTLE.HOOK_PIN_UP_LP := W#16#0;
   S_SHUTTLE.HOOK_PIN_DOWN_LP := W#16#0;
   S_SHUTTLE.DAECHA_LOCK_ADV_LP := W#16#0;
   S_SHUTTLE.DAECHA_LOCK_RET_LP := W#16#0;
   S_SHUTTLE.ELE_ADV_LP := W#16#0;
   S_SHUTTLE.ELE_RET_LP := W#16#0;
   S_SHUTTLE.AIR_ELE_ADV_LP := W#16#0;
   S_SHUTTLE.AIR_ELE_RET_LP := W#16#0;
   S_SHUTTLE.SP_WORD19 := W#16#0;
   S_SHUTTLE.SP_WORD20 := W#16#0;
   S_SHUTTLE.LM_DC_PIN_UP_LP := W#16#0;
   S_SHUTTLE.LM_DC_PIN_DOWN_LP := W#16#0;
   S_SHUTTLE.LM_DC_1ST_CLAMP1_ADV_LP := W#16#0;
   S_SHUTTLE.LM_DC_1ST_CLAMP1_RET_LP := W#16#0;
   S_SHUTTLE.LM_DC_1ST_CLAMP2_ADV_LP := W#16#0;
   S_SHUTTLE.LM_DC_1ST_CLAMP2_RET_LP := W#16#0;
   S_SHUTTLE.LM_DC_1ST_CLAMP3_ADV_LP := W#16#0;
   S_SHUTTLE.LM_DC_1ST_CLAMP3_RET_LP := W#16#0;
   S_SHUTTLE.LM_DC_1ST_CLAMP4_ADV_LP := W#16#0;
   S_SHUTTLE.LM_DC_1ST_CLAMP4_RET_LP := W#16#0;
   S_SHUTTLE.LM_DC_2ND_CLAMP1_ADV_LP := W#16#0;
   S_SHUTTLE.LM_DC_2ND_CLAMP1_RET_LP := W#16#0;
   S_SHUTTLE.LM_DC_2ND_CLAMP2_ADV_LP := W#16#0;
   S_SHUTTLE.LM_DC_2ND_CLAMP2_RET_LP := W#16#0;
   S_SHUTTLE.LM_DC_2ND_CLAMP3_ADV_LP := W#16#0;
   S_SHUTTLE.LM_DC_2ND_CLAMP3_RET_LP := W#16#0;
   S_SHUTTLE.LM_DC_2ND_CLAMP4_ADV_LP := W#16#0;
   S_SHUTTLE.LM_DC_2ND_CLAMP4_RET_LP := W#16#0;
   S_SHUTTLE.LM_DC_2ND_CLAMP5_ADV_LP := W#16#0;
   S_SHUTTLE.LM_DC_2ND_CLAMP5_RET_LP := W#16#0;
   S_SHUTTLE.LM_DC_DR_STK_PIN_UP_LP := W#16#0;
   S_SHUTTLE.LM_DC_DR_STK_PIN_DOWN_LP := W#16#0;
   S_SHUTTLE.LM_DC_OTR_CLAMP_ADV_LP := W#16#0;
   S_SHUTTLE.LM_DC_OTR_CLAMP_RET_LP := W#16#0;
   S_SHUTTLE.LM_DC_ASSY_CLAMP_ADV_LP := W#16#0;
   S_SHUTTLE.LM_DC_ASSY_CLAMP_RET_LP := W#16#0;
   S_SHUTTLE.LM_DC_FF_PIN_UP_LP := W#16#0;
   S_SHUTTLE.LM_DC_FF_PIN_DOWN_LP := W#16#0;
   S_SHUTTLE.LM_DC_FF_CLAMP_ADV_LP := W#16#0;
   S_SHUTTLE.LM_DC_FF_CLAMP_RET_LP := W#16#0;
   S_SHUTTLE.LM_DC_2ND_CLAMP6_ADV_LP := W#16#0;
   S_SHUTTLE.LM_DC_2ND_CLAMP6_RET_LP := W#16#0;
   S_SHUTTLE.LM_DC_2ND_CLAMP7_ADV_LP := W#16#0;
   S_SHUTTLE.LM_DC_2ND_CLAMP7_RET_LP := W#16#0;
   S_SHUTTLE.LM_DC_1ST_CLAMP5_ADV_LP := W#16#0;
   S_SHUTTLE.LM_DC_1ST_CLAMP5_RET_LP := W#16#0;
   S_SHUTTLE.SP_WORD68 := W#16#0;
   S_SHUTTLE.SP_WORD69 := W#16#0;
   S_SHUTTLE.SP_WORD70 := W#16#0;
   S_SHUTTLE.SP_WORD71 := W#16#0;
   S_SHUTTLE.TL_DC_PIN_UP_LP := W#16#0;
   S_SHUTTLE.TL_DC_PIN_DOWN_LP := W#16#0;
   S_SHUTTLE.TL_DC_LATCH1_ADV_LP := W#16#0;
   S_SHUTTLE.TL_DC_LATCH1_RET_LP := W#16#0;
   S_SHUTTLE.TL_DC_LATCH2_ADV_LP := W#16#0;
   S_SHUTTLE.TL_DC_LATCH2_RET_LP := W#16#0;
   S_SHUTTLE.TL_DC_1ST_CLAMP1_ADV_LP := W#16#0;
   S_SHUTTLE.TL_DC_1ST_CLAMP1_RET_LP := W#16#0;
   S_SHUTTLE.TL_DC_1ST_CLAMP2_ADV_LP := W#16#0;
   S_SHUTTLE.TL_DC_1ST_CLAMP2_RET_LP := W#16#0;
   S_SHUTTLE.TL_DC_1ST_CLAMP3_ADV_LP := W#16#0;
   S_SHUTTLE.TL_DC_1ST_CLAMP3_RET_LP := W#16#0;
   S_SHUTTLE.TL_DC_2ND_CLAMP1_ADV_LP := W#16#0;
   S_SHUTTLE.TL_DC_2ND_CLAMP1_RET_LP := W#16#0;
   S_SHUTTLE.TL_DC_2ND_CLAMP2_ADV_LP := W#16#0;
   S_SHUTTLE.TL_DC_2ND_CLAMP2_RET_LP := W#16#0;
   S_SHUTTLE.TL_DC_U261_ADV_LP := W#16#0;
   S_SHUTTLE.TL_DC_U261_RET_LP := W#16#0;
   S_SHUTTLE.TL_DC_U261_CLAMP_ADV_LP := W#16#0;
   S_SHUTTLE.TL_DC_U261_CLAMP_RET_LP := W#16#0;
   S_SHUTTLE.TL_DC_U269_UP_LP := W#16#0;
   S_SHUTTLE.TL_DC_U269_DOWN_LP := W#16#0;
   S_SHUTTLE.TL_DC_U269_CLAMP_ADV_LP := W#16#0;
   S_SHUTTLE.TL_DC_U269_CLAMP_RET_LP := W#16#0;
   S_SHUTTLE.TL_DC_3RD_CLAMP_ADV_LP := W#16#0;
   S_SHUTTLE.TL_DC_3RD_CLAMP_RET_LP := W#16#0;
   S_SHUTTLE.TL_DC_U262_1_UP_LP := W#16#0;
   S_SHUTTLE.TL_DC_U262_1_DOWN_LP := W#16#0;
   S_SHUTTLE.TL_DC_U262_1_ADV_LP := W#16#0;
   S_SHUTTLE.TL_DC_U262_1_RET_LP := W#16#0;
   S_SHUTTLE.TL_DC_U262_1_CLP_ADV_LP := W#16#0;
   S_SHUTTLE.TL_DC_U262_1_CLP_RET_LP := W#16#0;
   S_SHUTTLE.TL_DC_U261_2_CLP_ADV_LP := W#16#0;
   S_SHUTTLE.TL_DC_U261_2_CLP_RET_LP := W#16#0;
   S_SHUTTLE.SP_WORD106 := W#16#0;
   S_SHUTTLE.SP_WORD107 := W#16#0;
   S_SHUTTLE.SP_WORD108 := W#16#0;
   S_SHUTTLE.SP_WORD109 := W#16#0;
   S_SHUTTLE.SP_WORD110 := W#16#0;
   S_SHUTTLE.SP_WORD111 := W#16#0;
   S_702.M_AUTO_SEL := FALSE;
   S_702.M_MANUAL_SEL := FALSE;
   S_702.M_READY_PB := FALSE;
   S_702.M_AUTO_RUN_PB := FALSE;
   S_702.M_WORK_COMP_SET_PB := FALSE;
   S_702.M_WORK_COMP_RST_PB := FALSE;
   S_702.M_HOME_POS_PB := FALSE;
   S_702.M_TIP_DRESS_PB := FALSE;
   S_702.HOOK_PIN_SEL := FALSE;
   S_702.DAECHA_LOCK_SEL := FALSE;
   S_702.DAECHA_LOCK_UP_DN_SEL := FALSE;
   S_702.AIR_ELE_SEL := FALSE;
   S_702.EJECT_SEL := FALSE;
   S_702.STOPPER_SER := FALSE;
   S_702.DAECHA_CLAMP_SEL := FALSE;
   S_702.SHOCK_ABSORBER_SEL := FALSE;
   S_702.DAECHA_IN_SEL := FALSE;
   S_702.DAECHA_OUT_SEL := FALSE;
   S_702.SPARE19 := FALSE;
   S_702.SPARE20 := FALSE;
   S_702.SPARE21 := FALSE;
   S_702.SPARE22 := FALSE;
   S_702.SPARE23 := FALSE;
   S_702.SPARE24 := FALSE;
   S_702.LINE_EMPTY_SS := FALSE;
   S_702.OUT_TRV_BT_ON_PB := FALSE;
   S_702.SPARE27 := FALSE;
   S_702.SPARE28 := FALSE;
   S_702.SPARE29 := FALSE;
   S_702.SPARE30 := FALSE;
   S_702.M_ADV_PB := FALSE;
   S_702.M_RET_PB := FALSE;
   S_702.LM_DC_PIN_SEL := FALSE;
   S_702.LM_DC_1ST_CLAMP1_SEL := FALSE;
   S_702.LM_DC_1ST_CLAMP2_SEL := FALSE;
   S_702.LM_DC_1ST_CLAMP3_SEL := FALSE;
   S_702.LM_DC_1ST_CLAMP4_SEL := FALSE;
   S_702.LM_DC_2ND_CLAMP1_SEL := FALSE;
   S_702.LM_DC_2ND_CLAMP2_SEL := FALSE;
   S_702.LM_DC_2ND_CLAMP3_SEL := FALSE;
   S_702.LM_DC_2ND_CLAMP4_SEL := FALSE;
   S_702.LM_DC_2ND_CLAMP5_SEL := FALSE;
   S_702.LM_DC_DR_STK_PIN_SEL := FALSE;
   S_702.LM_DC_OTR_CLAMP_SEL := FALSE;
   S_702.LM_DC_ASSY_CLAMP_SEL := FALSE;
   S_702.LM_DC_FF_PIN_SEL := FALSE;
   S_702.LM_DC_FF_CLAMP_SEL := FALSE;
   S_702.LM_DC_2ND_CLAMP6_SEL := FALSE;
   S_702.SPARE50 := FALSE;
   S_702.SPARE51 := FALSE;
   S_702.SPARE52 := FALSE;
   S_702.SPARE53 := FALSE;
   S_702.SPARE54 := FALSE;
   S_702.SPARE55 := FALSE;
   S_702.SPARE56 := FALSE;
   S_702.SPARE57 := FALSE;
   S_702.SPARE58 := FALSE;
   S_702.SPARE59 := FALSE;
   S_702.SPARE60 := FALSE;
   S_702.SPARE61 := FALSE;
   S_702.SPARE62 := FALSE;
   S_702.SPARE63 := FALSE;
   S_702.LM_DC_M_ADV_PB := FALSE;
   S_702.LM_DC_M_RET_PB := FALSE;
   S_702.TL_DC_PIN_SEL := FALSE;
   S_702.TL_DC_LATCH1_SEL := FALSE;
   S_702.TL_DC_1ST_CLAMP_SEL := FALSE;
   S_702.TL_DC_2ND_CLAMP_SEL := FALSE;
   S_702.TL_DC_U261_SEL := FALSE;
   S_702.TL_DC_U261_CLAMP_SEL := FALSE;
   S_702.TL_DC_U269_UP_DN_SEL := FALSE;
   S_702.TL_DC_U269_CLAMP_SEL := FALSE;
   S_702.TL_DC_3RD_CLAMP_SEL := FALSE;
   S_702.TL_DC_U262_1_UP_DN_SEL := FALSE;
   S_702.TL_DC_U262_1_SEL := FALSE;
   S_702.TL_DC_U262_1_CLAMP_SEL := FALSE;
   S_702.TL_DC_U261_2_CLAMP_SEL := FALSE;
   S_702.SPARE79 := FALSE;
   S_702.SPARE80 := FALSE;
   S_702.SPARE81 := FALSE;
   S_702.SPARE82 := FALSE;
   S_702.SPARE83 := FALSE;
   S_702.SPARE84 := FALSE;
   S_702.SPARE85 := FALSE;
   S_702.SPARE86 := FALSE;
   S_702.SPARE87 := FALSE;
   S_702.SPARE88 := FALSE;
   S_702.SPARE89 := FALSE;
   S_702.SPARE90 := FALSE;
   S_702.SPARE91 := FALSE;
   S_702.SPARE92 := FALSE;
   S_702.SPARE93 := FALSE;
   S_702.SPARE94 := FALSE;
   S_702.SPARE95 := FALSE;
   S_702.TL_DC_M_ADV_PB := FALSE;
   S_702.TL_DC_M_RET_PB := FALSE;
   S_702.SPARE98 := FALSE;
   S_702.SPARE99 := FALSE;
   S_702.SPARE100 := FALSE;
   S_702.SPARE101 := FALSE;
   S_702.SPARE102 := FALSE;
   S_702.SPARE103 := FALSE;
   S_702.SPARE104 := FALSE;
   S_702.SPARE105 := FALSE;
   S_702.SPARE106 := FALSE;
   S_702.SPARE107 := FALSE;
   S_702.SPARE108 := FALSE;
   S_702.SPARE109 := FALSE;
   S_702.SPARE110 := FALSE;
   S_702.SPARE111 := FALSE;
   S_702.SPARE112 := FALSE;
   S_702.SPARE113 := FALSE;
   S_702.SPARE114 := FALSE;
   S_702.SPARE115 := FALSE;
   S_702.SPARE116 := FALSE;
   S_702.SPARE117 := FALSE;
   S_702.SPARE118 := FALSE;
   S_702.SPARE119 := FALSE;
   S_702.SPARE120 := FALSE;
   S_702.SPARE121 := FALSE;
   S_702.SPARE122 := FALSE;
   S_702.SPARE123 := FALSE;
   S_702.SPARE124 := FALSE;
   S_702.SPARE125 := FALSE;
   S_702.SPARE126 := FALSE;
   S_702.SPARE127 := FALSE;
   S_702.SPARE128 := FALSE;
   S_702.SPARE129 := FALSE;
   S_702.SPARE130 := FALSE;
   S_702.SPARE131 := FALSE;
   S_702.SPARE132 := FALSE;
   S_702.SPARE133 := FALSE;
   S_702.SPARE134 := FALSE;
   S_702.SPARE135 := FALSE;
   S_702.SPARE136 := FALSE;
   S_702.SPARE137 := FALSE;
   S_702.SPARE138 := FALSE;
   S_702.SPARE139 := FALSE;
   S_702.SPARE140 := FALSE;
   S_702.SPARE141 := FALSE;
   S_702.SPARE142 := FALSE;
   S_702.SPARE143 := FALSE;
   S_702.SPARE144 := FALSE;
   S_702.SPARE145 := FALSE;
   S_702.SPARE146 := FALSE;
   S_702.SPARE147 := FALSE;
   S_702.SPARE148 := FALSE;
   S_702.SPARE149 := FALSE;
   S_702.SPARE150 := FALSE;
   S_702.SPARE151 := FALSE;
   S_702.SPARE152 := FALSE;
   S_702.SPARE153 := FALSE;
   S_702.SPARE154 := FALSE;
   S_702.SPARE155 := FALSE;
   S_702.SPARE156 := FALSE;
   S_702.SPARE157 := FALSE;
   S_702.SPARE158 := FALSE;
   S_702.SPARE159 := FALSE;
   S_702.SPARE160 := FALSE;
   S_702.SPARE161 := FALSE;
   S_702.HOOK_PIN_UP_LP := W#16#0;
   S_702.HOOK_PIN_DOWN_LP := W#16#0;
   S_702.DAECHA_LOCK_ADV_LP := W#16#0;
   S_702.DAECHA_LOCK_RET_LP := W#16#0;
   S_702.DAECHA_LOCK_UP_LP := W#16#0;
   S_702.DAECHA_LOCK_DOWN_LP := W#16#0;
   S_702.ELE_ADV_LP := W#16#0;
   S_702.ELE_RET_LP := W#16#0;
   S_702.AIR_ELE_ADV_LP := W#16#0;
   S_702.AIR_ELE_RET_LP := W#16#0;
   S_702.LM_DC_PIN_UP_LP := W#16#0;
   S_702.LM_DC_PIN_DOWN_LP := W#16#0;
   S_702.LM_DC_1ST_CLAMP1_ADV_LP := W#16#0;
   S_702.LM_DC_1ST_CLAMP1_RET_LP := W#16#0;
   S_702.LM_DC_1ST_CLAMP2_ADV_LP := W#16#0;
   S_702.LM_DC_1ST_CLAMP2_RET_LP := W#16#0;
   S_702.LM_DC_1ST_CLAMP3_ADV_LP := W#16#0;
   S_702.LM_DC_1ST_CLAMP3_RET_LP := W#16#0;
   S_702.LM_DC_1ST_CLAMP4_ADV_LP := W#16#0;
   S_702.LM_DC_1ST_CLAMP4_RET_LP := W#16#0;
   S_702.LM_DC_2ND_CLAMP1_ADV_LP := W#16#0;
   S_702.LM_DC_2ND_CLAMP1_RET_LP := W#16#0;
   S_702.LM_DC_2ND_CLAMP2_ADV_LP := W#16#0;
   S_702.LM_DC_2ND_CLAMP2_RET_LP := W#16#0;
   S_702.LM_DC_2ND_CLAMP3_ADV_LP := W#16#0;
   S_702.LM_DC_2ND_CLAMP3_RET_LP := W#16#0;
   S_702.LM_DC_2ND_CLAMP4_ADV_LP := W#16#0;
   S_702.LM_DC_2ND_CLAMP4_RET_LP := W#16#0;
   S_702.LM_DC_2ND_CLAMP5_ADV_LP := W#16#0;
   S_702.LM_DC_2ND_CLAMP5_RET_LP := W#16#0;
   S_702.LM_DC_DR_STK_PIN_UP_LP := W#16#0;
   S_702.LM_DC_DR_STK_PIN_DOWN_LP := W#16#0;
   S_702.LM_DC_OTR_CLAMP_ADV_LP := W#16#0;
   S_702.LM_DC_OTR_CLAMP_RET_LP := W#16#0;
   S_702.LM_DC_ASSY_CLAMP_ADV_LP := W#16#0;
   S_702.LM_DC_ASSY_CLAMP_RET_LP := W#16#0;
   S_702.LM_DC_FF_PIN_UP_LP := W#16#0;
   S_702.LM_DC_FF_PIN_DOWN_LP := W#16#0;
   S_702.LM_DC_FF_CLAMP_ADV_LP := W#16#0;
   S_702.LM_DC_FF_CLAMP_RET_LP := W#16#0;
   S_702.LM_DC_2ND_CLAMP6_ADV_LP := W#16#0;
   S_702.LM_DC_2ND_CLAMP6_RET_LP := W#16#0;
   S_702.LM_DC_2ND_CLAMP7_ADV_LP := W#16#0;
   S_702.LM_DC_2ND_CLAMP7_RET_LP := W#16#0;
   S_702.LM_DC_1ST_CLAMP5_ADV_LP := W#16#0;
   S_702.LM_DC_1ST_CLAMP5_RET_LP := W#16#0;
   S_702.EJECT_UP_LP := W#16#0;
   S_702.EJECT_DOWN_LP := W#16#0;
   S_702.STOPPER_ADV_LP := W#16#0;
   S_702.STOPPER_RET_LP := W#16#0;
   S_702.TL_DC_PIN_UP_LP := W#16#0;
   S_702.TL_DC_PIN_DOWN_LP := W#16#0;
   S_702.TL_DC_LATCH1_ADV_LP := W#16#0;
   S_702.TL_DC_LATCH1_RET_LP := W#16#0;
   S_702.TL_DC_LATCH2_ADV_LP := W#16#0;
   S_702.TL_DC_LATCH2_RET_LP := W#16#0;
   S_702.TL_DC_1ST_CLAMP1_ADV_LP := W#16#0;
   S_702.TL_DC_1ST_CLAMP1_RET_LP := W#16#0;
   S_702.TL_DC_1ST_CLAMP2_ADV_LP := W#16#0;
   S_702.TL_DC_1ST_CLAMP2_RET_LP := W#16#0;
   S_702.TL_DC_1ST_CLAMP3_ADV_LP := W#16#0;
   S_702.TL_DC_1ST_CLAMP3_RET_LP := W#16#0;
   S_702.TL_DC_2ND_CLAMP1_ADV_LP := W#16#0;
   S_702.TL_DC_2ND_CLAMP1_RET_LP := W#16#0;
   S_702.TL_DC_2ND_CLAMP2_ADV_LP := W#16#0;
   S_702.TL_DC_2ND_CLAMP2_RET_LP := W#16#0;
   S_702.TL_DC_U261_ADV_LP := W#16#0;
   S_702.TL_DC_U261_RET_LP := W#16#0;
   S_702.TL_DC_U261_CLAMP_ADV_LP := W#16#0;
   S_702.TL_DC_U261_CLAMP_RET_LP := W#16#0;
   S_702.TL_DC_U269_UP_LP := W#16#0;
   S_702.TL_DC_U269_DOWN_LP := W#16#0;
   S_702.TL_DC_U269_CLAMP_ADV_LP := W#16#0;
   S_702.TL_DC_U269_CLAMP_RET_LP := W#16#0;
   S_702.TL_DC_3RD_CLAMP_ADV_LP := W#16#0;
   S_702.TL_DC_3RD_CLAMP_RET_LP := W#16#0;
   S_702.TL_DC_U262_1_UP_LP := W#16#0;
   S_702.TL_DC_U262_1_DOWN_LP := W#16#0;
   S_702.TL_DC_U262_1_ADV_LP := W#16#0;
   S_702.TL_DC_U262_1_RET_LP := W#16#0;
   S_702.TL_DC_U262_1_CLP_ADV_LP := W#16#0;
   S_702.TL_DC_U262_1_CLP_RET_LP := W#16#0;
   S_702.TL_DC_U261_2_CLP_ADV_LP := W#16#0;
   S_702.TL_DC_U261_2_CLP_RET_LP := W#16#0;
   S_702.SP_WORD106 := W#16#0;
   S_702.SP_WORD107 := W#16#0;
   S_702.DAECHA_CLAMP_ADV_LP := W#16#0;
   S_702.DAECHA_CLAMP_RET_LP := W#16#0;
   S_702.SHOCK_ABSORBER_ADV_LP := W#16#0;
   S_702.SHOCK_ABSORBER_RET_LP := W#16#0;
   S_703.M_AUTO_SEL := FALSE;
   S_703.M_MANUAL_SEL := FALSE;
   S_703.M_READY_PB := FALSE;
   S_703.M_AUTO_RUN_PB := FALSE;
   S_703.M_WORK_COMP_SET_PB := FALSE;
   S_703.M_WORK_COMP_RST_PB := FALSE;
   S_703.M_HOME_POS_PB := FALSE;
   S_703.M_TIP_DRESS_PB := FALSE;
   S_703.HOOK_PIN_SEL := FALSE;
   S_703.DAECHA_LOCK_SEL := FALSE;
   S_703.ELE_SEL := FALSE;
   S_703.SPARE12 := FALSE;
   S_703.SPARE13 := FALSE;
   S_703.SPARE14 := FALSE;
   S_703.SPARE15 := FALSE;
   S_703.SPARE16 := FALSE;
   S_703.SPARE17 := FALSE;
   S_703.SPARE18 := FALSE;
   S_703.SPARE19 := FALSE;
   S_703.SPARE20 := FALSE;
   S_703.SPARE21 := FALSE;
   S_703.SPARE22 := FALSE;
   S_703.SPARE23 := FALSE;
   S_703.SPARE24 := FALSE;
   S_703.SPARE25 := FALSE;
   S_703.SPARE26 := FALSE;
   S_703.SPARE27 := FALSE;
   S_703.SPARE28 := FALSE;
   S_703.SPARE29 := FALSE;
   S_703.SPARE30 := FALSE;
   S_703.M_ADV_PB := FALSE;
   S_703.M_RET_PB := FALSE;
   S_703.LM_DC_PIN_SEL := FALSE;
   S_703.LM_DC_1ST_CLAMP1_SEL := FALSE;
   S_703.LM_DC_1ST_CLAMP2_SEL := FALSE;
   S_703.LM_DC_1ST_CLAMP3_SEL := FALSE;
   S_703.LM_DC_1ST_CLAMP4_SEL := FALSE;
   S_703.LM_DC_2ND_CLAMP1_SEL := FALSE;
   S_703.LM_DC_2ND_CLAMP2_SEL := FALSE;
   S_703.LM_DC_2ND_CLAMP3_SEL := FALSE;
   S_703.LM_DC_2ND_CLAMP4_SEL := FALSE;
   S_703.LM_DC_2ND_CLAMP5_SEL := FALSE;
   S_703.LM_DC_DR_STK_PIN_SEL := FALSE;
   S_703.LM_DC_OTR_CLAMP_SEL := FALSE;
   S_703.LM_DC_ASSY_CLAMP_SEL := FALSE;
   S_703.LM_DC_FF_PIN_SEL := FALSE;
   S_703.LM_DC_FF_CLAMP_SEL := FALSE;
   S_703.LM_DC_2ND_CLAMP6_SEL := FALSE;
   S_703.SPARE50 := FALSE;
   S_703.SPARE51 := FALSE;
   S_703.SPARE52 := FALSE;
   S_703.SPARE53 := FALSE;
   S_703.SPARE54 := FALSE;
   S_703.SPARE55 := FALSE;
   S_703.SPARE56 := FALSE;
   S_703.SPARE57 := FALSE;
   S_703.SPARE58 := FALSE;
   S_703.SPARE59 := FALSE;
   S_703.SPARE60 := FALSE;
   S_703.SPARE61 := FALSE;
   S_703.SPARE62 := FALSE;
   S_703.SPARE63 := FALSE;
   S_703.LM_DC_M_ADV_PB := FALSE;
   S_703.LM_DC_M_RET_PB := FALSE;
   S_703.TL_DC_PIN_SEL := FALSE;
   S_703.TL_DC_LATCH1_SEL := FALSE;
   S_703.TL_DC_1ST_CLAMP_SEL := FALSE;
   S_703.TL_DC_2ND_CLAMP_SEL := FALSE;
   S_703.TL_DC_U261_SEL := FALSE;
   S_703.TL_DC_U261_CLAMP_SEL := FALSE;
   S_703.TL_DC_U269_UP_DN_SEL := FALSE;
   S_703.TL_DC_U269_CLAMP_SEL := FALSE;
   S_703.TL_DC_3RD_CLAMP_SEL := FALSE;
   S_703.TL_DC_U262_1_UP_DN_SEL := FALSE;
   S_703.TL_DC_U262_1_SEL := FALSE;
   S_703.TL_DC_U262_1_CLAMP_SEL := FALSE;
   S_703.TL_DC_U261_2_CLAMP_SEL := FALSE;
   S_703.SPARE79 := FALSE;
   S_703.SPARE80 := FALSE;
   S_703.SPARE81 := FALSE;
   S_703.SPARE82 := FALSE;
   S_703.SPARE83 := FALSE;
   S_703.SPARE84 := FALSE;
   S_703.SPARE85 := FALSE;
   S_703.SPARE86 := FALSE;
   S_703.SPARE87 := FALSE;
   S_703.SPARE88 := FALSE;
   S_703.SPARE89 := FALSE;
   S_703.SPARE90 := FALSE;
   S_703.SPARE91 := FALSE;
   S_703.SPARE92 := FALSE;
   S_703.SPARE93 := FALSE;
   S_703.SPARE94 := FALSE;
   S_703.SPARE95 := FALSE;
   S_703.TL_DC_M_ADV_PB := FALSE;
   S_703.TL_DC_M_RET_PB := FALSE;
   S_703.SPARE98 := FALSE;
   S_703.SPARE99 := FALSE;
   S_703.SPARE100 := FALSE;
   S_703.SPARE101 := FALSE;
   S_703.SPARE102 := FALSE;
   S_703.SPARE103 := FALSE;
   S_703.SPARE104 := FALSE;
   S_703.SPARE105 := FALSE;
   S_703.SPARE106 := FALSE;
   S_703.SPARE107 := FALSE;
   S_703.SPARE108 := FALSE;
   S_703.SPARE109 := FALSE;
   S_703.SPARE110 := FALSE;
   S_703.SPARE111 := FALSE;
   S_703.SPARE112 := FALSE;
   S_703.SPARE113 := FALSE;
   S_703.SPARE114 := FALSE;
   S_703.SPARE115 := FALSE;
   S_703.SPARE116 := FALSE;
   S_703.SPARE117 := FALSE;
   S_703.SPARE118 := FALSE;
   S_703.SPARE119 := FALSE;
   S_703.SPARE120 := FALSE;
   S_703.SPARE121 := FALSE;
   S_703.SPARE122 := FALSE;
   S_703.SPARE123 := FALSE;
   S_703.SPARE124 := FALSE;
   S_703.SPARE125 := FALSE;
   S_703.SPARE126 := FALSE;
   S_703.SPARE127 := FALSE;
   S_703.SPARE128 := FALSE;
   S_703.SPARE129 := FALSE;
   S_703.SPARE130 := FALSE;
   S_703.SPARE131 := FALSE;
   S_703.SPARE132 := FALSE;
   S_703.SPARE133 := FALSE;
   S_703.SPARE134 := FALSE;
   S_703.SPARE135 := FALSE;
   S_703.SPARE136 := FALSE;
   S_703.SPARE137 := FALSE;
   S_703.SPARE138 := FALSE;
   S_703.SPARE139 := FALSE;
   S_703.SPARE140 := FALSE;
   S_703.SPARE141 := FALSE;
   S_703.SPARE142 := FALSE;
   S_703.SPARE143 := FALSE;
   S_703.SPARE144 := FALSE;
   S_703.SPARE145 := FALSE;
   S_703.SPARE146 := FALSE;
   S_703.SPARE147 := FALSE;
   S_703.SPARE148 := FALSE;
   S_703.SPARE149 := FALSE;
   S_703.SPARE150 := FALSE;
   S_703.SPARE151 := FALSE;
   S_703.SPARE152 := FALSE;
   S_703.SPARE153 := FALSE;
   S_703.SPARE154 := FALSE;
   S_703.SPARE155 := FALSE;
   S_703.SPARE156 := FALSE;
   S_703.SPARE157 := FALSE;
   S_703.SPARE158 := FALSE;
   S_703.SPARE159 := FALSE;
   S_703.SPARE160 := FALSE;
   S_703.SPARE161 := FALSE;
   S_703.HOOK_PIN_UP_LP := W#16#0;
   S_703.HOOK_PIN_DOWN_LP := W#16#0;
   S_703.DAECHA_LOCK_ADV_LP := W#16#0;
   S_703.DAECHA_LOCK_RET_LP := W#16#0;
   S_703.ELE_ADV_LP := W#16#0;
   S_703.ELE_RET_LP := W#16#0;
   S_703.AIR_ELE_ADV_LP := W#16#0;
   S_703.AIR_ELE_RET_LP := W#16#0;
   S_703.SP_WORD19 := W#16#0;
   S_703.SP_WORD20 := W#16#0;
   S_703.LM_DC_PIN_UP_LP := W#16#0;
   S_703.LM_DC_PIN_DOWN_LP := W#16#0;
   S_703.LM_DC_1ST_CLAMP1_ADV_LP := W#16#0;
   S_703.LM_DC_1ST_CLAMP1_RET_LP := W#16#0;
   S_703.LM_DC_1ST_CLAMP2_ADV_LP := W#16#0;
   S_703.LM_DC_1ST_CLAMP2_RET_LP := W#16#0;
   S_703.LM_DC_1ST_CLAMP3_ADV_LP := W#16#0;
   S_703.LM_DC_1ST_CLAMP3_RET_LP := W#16#0;
   S_703.LM_DC_1ST_CLAMP4_ADV_LP := W#16#0;
   S_703.LM_DC_1ST_CLAMP4_RET_LP := W#16#0;
   S_703.LM_DC_2ND_CLAMP1_ADV_LP := W#16#0;
   S_703.LM_DC_2ND_CLAMP1_RET_LP := W#16#0;
   S_703.LM_DC_2ND_CLAMP2_ADV_LP := W#16#0;
   S_703.LM_DC_2ND_CLAMP2_RET_LP := W#16#0;
   S_703.LM_DC_2ND_CLAMP3_ADV_LP := W#16#0;
   S_703.LM_DC_2ND_CLAMP3_RET_LP := W#16#0;
   S_703.LM_DC_2ND_CLAMP4_ADV_LP := W#16#0;
   S_703.LM_DC_2ND_CLAMP4_RET_LP := W#16#0;
   S_703.LM_DC_2ND_CLAMP5_ADV_LP := W#16#0;
   S_703.LM_DC_2ND_CLAMP5_RET_LP := W#16#0;
   S_703.LM_DC_DR_STK_PIN_UP_LP := W#16#0;
   S_703.LM_DC_DR_STK_PIN_DOWN_LP := W#16#0;
   S_703.LM_DC_OTR_CLAMP_ADV_LP := W#16#0;
   S_703.LM_DC_OTR_CLAMP_RET_LP := W#16#0;
   S_703.LM_DC_ASSY_CLAMP_ADV_LP := W#16#0;
   S_703.LM_DC_ASSY_CLAMP_RET_LP := W#16#0;
   S_703.LM_DC_FF_PIN_UP_LP := W#16#0;
   S_703.LM_DC_FF_PIN_DOWN_LP := W#16#0;
   S_703.LM_DC_FF_CLAMP_ADV_LP := W#16#0;
   S_703.LM_DC_FF_CLAMP_RET_LP := W#16#0;
   S_703.LM_DC_2ND_CLAMP6_ADV_LP := W#16#0;
   S_703.LM_DC_2ND_CLAMP6_RET_LP := W#16#0;
   S_703.LM_DC_2ND_CLAMP7_ADV_LP := W#16#0;
   S_703.LM_DC_2ND_CLAMP7_RET_LP := W#16#0;
   S_703.LM_DC_1ST_CLAMP5_ADV_LP := W#16#0;
   S_703.LM_DC_1ST_CLAMP5_RET_LP := W#16#0;
   S_703.SP_WORD68 := W#16#0;
   S_703.SP_WORD69 := W#16#0;
   S_703.SP_WORD70 := W#16#0;
   S_703.SP_WORD71 := W#16#0;
   S_703.TL_DC_PIN_UP_LP := W#16#0;
   S_703.TL_DC_PIN_DOWN_LP := W#16#0;
   S_703.TL_DC_LATCH1_ADV_LP := W#16#0;
   S_703.TL_DC_LATCH1_RET_LP := W#16#0;
   S_703.TL_DC_LATCH2_ADV_LP := W#16#0;
   S_703.TL_DC_LATCH2_RET_LP := W#16#0;
   S_703.TL_DC_1ST_CLAMP1_ADV_LP := W#16#0;
   S_703.TL_DC_1ST_CLAMP1_RET_LP := W#16#0;
   S_703.TL_DC_1ST_CLAMP2_ADV_LP := W#16#0;
   S_703.TL_DC_1ST_CLAMP2_RET_LP := W#16#0;
   S_703.TL_DC_1ST_CLAMP3_ADV_LP := W#16#0;
   S_703.TL_DC_1ST_CLAMP3_RET_LP := W#16#0;
   S_703.TL_DC_2ND_CLAMP1_ADV_LP := W#16#0;
   S_703.TL_DC_2ND_CLAMP1_RET_LP := W#16#0;
   S_703.TL_DC_2ND_CLAMP2_ADV_LP := W#16#0;
   S_703.TL_DC_2ND_CLAMP2_RET_LP := W#16#0;
   S_703.TL_DC_U261_ADV_LP := W#16#0;
   S_703.TL_DC_U261_RET_LP := W#16#0;
   S_703.TL_DC_U261_CLAMP_ADV_LP := W#16#0;
   S_703.TL_DC_U261_CLAMP_RET_LP := W#16#0;
   S_703.TL_DC_U269_UP_LP := W#16#0;
   S_703.TL_DC_U269_DOWN_LP := W#16#0;
   S_703.TL_DC_U269_CLAMP_ADV_LP := W#16#0;
   S_703.TL_DC_U269_CLAMP_RET_LP := W#16#0;
   S_703.TL_DC_3RD_CLAMP_ADV_LP := W#16#0;
   S_703.TL_DC_3RD_CLAMP_RET_LP := W#16#0;
   S_703.TL_DC_U262_1_UP_LP := W#16#0;
   S_703.TL_DC_U262_1_DOWN_LP := W#16#0;
   S_703.TL_DC_U262_1_ADV_LP := W#16#0;
   S_703.TL_DC_U262_1_RET_LP := W#16#0;
   S_703.TL_DC_U262_1_CLP_ADV_LP := W#16#0;
   S_703.TL_DC_U262_1_CLP_RET_LP := W#16#0;
   S_703.TL_DC_U261_2_CLP_ADV_LP := W#16#0;
   S_703.TL_DC_U261_2_CLP_RET_LP := W#16#0;
   S_703.SP_WORD106 := W#16#0;
   S_703.SP_WORD107 := W#16#0;
   S_703.SP_WORD108 := W#16#0;
   S_703.SP_WORD109 := W#16#0;
   S_703.SP_WORD110 := W#16#0;
   S_703.SP_WORD111 := W#16#0;
   S_704.M_AUTO_SEL := FALSE;
   S_704.M_MANUAL_SEL := FALSE;
   S_704.M_READY_PB := FALSE;
   S_704.M_AUTO_RUN_PB := FALSE;
   S_704.M_WORK_COMP_SET_PB := FALSE;
   S_704.M_WORK_COMP_RST_PB := FALSE;
   S_704.M_HOME_POS_PB := FALSE;
   S_704.M_708_L_R_BT_ERR_RST := FALSE;
   S_704.HOOK_PIN_SEL := FALSE;
   S_704.DAECHA_LOCK_SEL := FALSE;
   S_704.ELE_SEL := FALSE;
   S_704.FF_CLAMP_SEL := FALSE;
   S_704.SPARE13 := FALSE;
   S_704.SPARE14 := FALSE;
   S_704.SPARE15 := FALSE;
   S_704.SPARE16 := FALSE;
   S_704.SPARE17 := FALSE;
   S_704.SPARE18 := FALSE;
   S_704.SPARE19 := FALSE;
   S_704.SPARE20 := FALSE;
   S_704.SPARE21 := FALSE;
   S_704.SPARE22 := FALSE;
   S_704.SPARE23 := FALSE;
   S_704.SPARE24 := FALSE;
   S_704.SPARE25 := FALSE;
   S_704.SPARE26 := FALSE;
   S_704.SPARE27 := FALSE;
   S_704.SPARE28 := FALSE;
   S_704.SPARE29 := FALSE;
   S_704.SPARE30 := FALSE;
   S_704.M_ADV_PB := FALSE;
   S_704.M_RET_PB := FALSE;
   S_704.LM_DC_PIN_SEL := FALSE;
   S_704.LM_DC_1ST_CLAMP1_SEL := FALSE;
   S_704.LM_DC_1ST_CLAMP2_SEL := FALSE;
   S_704.LM_DC_1ST_CLAMP3_SEL := FALSE;
   S_704.LM_DC_1ST_CLAMP4_SEL := FALSE;
   S_704.LM_DC_2ND_CLAMP1_SEL := FALSE;
   S_704.LM_DC_2ND_CLAMP2_SEL := FALSE;
   S_704.LM_DC_2ND_CLAMP3_SEL := FALSE;
   S_704.LM_DC_2ND_CLAMP4_SEL := FALSE;
   S_704.LM_DC_2ND_CLAMP5_SEL := FALSE;
   S_704.LM_DC_DR_STK_PIN_SEL := FALSE;
   S_704.LM_DC_OTR_CLAMP_SEL := FALSE;
   S_704.LM_DC_ASSY_CLAMP_SEL := FALSE;
   S_704.LM_DC_FF_PIN_SEL := FALSE;
   S_704.LM_DC_FF_CLAMP_SEL := FALSE;
   S_704.LM_DC_2ND_CLAMP6_SEL := FALSE;
   S_704.SPARE50 := FALSE;
   S_704.SPARE51 := FALSE;
   S_704.SPARE52 := FALSE;
   S_704.SPARE53 := FALSE;
   S_704.SPARE54 := FALSE;
   S_704.SPARE55 := FALSE;
   S_704.SPARE56 := FALSE;
   S_704.SPARE57 := FALSE;
   S_704.SPARE58 := FALSE;
   S_704.SPARE59 := FALSE;
   S_704.SPARE60 := FALSE;
   S_704.SPARE61 := FALSE;
   S_704.SPARE62 := FALSE;
   S_704.SPARE63 := FALSE;
   S_704.LM_DC_M_ADV_PB := FALSE;
   S_704.LM_DC_M_RET_PB := FALSE;
   S_704.TL_DC_PIN_SEL := FALSE;
   S_704.TL_DC_LATCH1_SEL := FALSE;
   S_704.TL_DC_1ST_CLAMP_SEL := FALSE;
   S_704.TL_DC_2ND_CLAMP_SEL := FALSE;
   S_704.TL_DC_U261_SEL := FALSE;
   S_704.TL_DC_U261_CLAMP_SEL := FALSE;
   S_704.TL_DC_U269_UP_DN_SEL := FALSE;
   S_704.TL_DC_U269_CLAMP_SEL := FALSE;
   S_704.TL_DC_3RD_CLAMP_SEL := FALSE;
   S_704.TL_DC_U262_1_UP_DN_SEL := FALSE;
   S_704.TL_DC_U262_1_SEL := FALSE;
   S_704.TL_DC_U262_1_CLAMP_SEL := FALSE;
   S_704.TL_DC_U261_2_CLAMP_SEL := FALSE;
   S_704.SPARE79 := FALSE;
   S_704.SPARE80 := FALSE;
   S_704.SPARE81 := FALSE;
   S_704.SPARE82 := FALSE;
   S_704.SPARE83 := FALSE;
   S_704.SPARE84 := FALSE;
   S_704.SPARE85 := FALSE;
   S_704.SPARE86 := FALSE;
   S_704.SPARE87 := FALSE;
   S_704.SPARE88 := FALSE;
   S_704.SPARE89 := FALSE;
   S_704.SPARE90 := FALSE;
   S_704.SPARE91 := FALSE;
   S_704.SPARE92 := FALSE;
   S_704.SPARE93 := FALSE;
   S_704.SPARE94 := FALSE;
   S_704.SPARE95 := FALSE;
   S_704.TL_DC_M_ADV_PB := FALSE;
   S_704.TL_DC_M_RET_PB := FALSE;
   S_704.SPARE98 := FALSE;
   S_704.SPARE99 := FALSE;
   S_704.SPARE100 := FALSE;
   S_704.SPARE101 := FALSE;
   S_704.SPARE102 := FALSE;
   S_704.SPARE103 := FALSE;
   S_704.SPARE104 := FALSE;
   S_704.SPARE105 := FALSE;
   S_704.SPARE106 := FALSE;
